(* USED TO LATCH A BIT TO CLEAR DATA AFTER UPSTACK TEST MODE IS OFF *)
IF 	csp_transfer_upstacker_sensors.debug_active
THEN
	debug_active_bool := TRUE;
END_IF

IF 	debug_active_bool
	AND NOT csp_transfer_upstacker_sensors.debug_active
THEN
	debug_active_clear := TRUE;
	debug_active_bool := FALSE;
END_IF

dry_cycle_ftrig(CLK :=csp_case_main_services.dry_cycle_mode); // falling edge of dry cycle mode, clear upstacker counts on completion of dry cycle mode. 
cleanout_mode_ftrig(CLK :=csp_main_motorization.empty_command); // falling edge of clean out mode, clear upstacker counts on completion of dry cycle mode. 


(* CLEARS SHIFT REGISTER BITS DURING SIZE CHANGE *)
IF 	csp_main_accuchange.machine_empty
	OR debug_active_clear
	OR process_message_is_on(csp_case_virtualMaster.runout_complete)
	OR dry_cycle_ftrig.Q
	OR cleanout_mode_ftrig.Q
THEN
	stack_count := 0;
	stack_made := FALSE;
	stack_on_way_to_loader := FALSE;
	stack_at_loader := FALSE;
	First_cycle_after_dry := TRUE;
	debug_active_clear := FALSE;
END_IF

//Resets First_Cycle_After_Dry

IF 	First_Cycle_After_Dry
	AND csp_main_motorization_virtualManager.axis.actual_position > 355
	AND csp_main_motorization_virtualManager.axis.actual_position < 359
THEN
	First_Cycle_After_Dry := False;
END_IF


(* CLEARS STACK AT LOADER AND ON WAY TO LOADER IF CROSSPUSHER REJECT *)
IF 	csp_transfer_crosspusher.reject_running
THEN
	stack_on_way_to_loader := FALSE;
	stack_at_loader := FALSE;
END_IF


(* MANUAL REMOVAL OF STACK AT UPSTACKER *)
IF 	stack_removed_from_upstack_cbtn.value_from_hmi = HMI_BUTTON_STATUS_ON//command_button_is_pressed(stack_removed_from_upstack_cbtn) 
THEN
	stack_removed_from_upstack := TRUE;
ELSE
	stack_removed_from_upstack := FALSE;
END_IF

IF stack_removed_from_upstack
THEN
	stack_count := 0;
END_IF


(* CHECKS STACK COUNT AGAINST CASE PATTERN COUNT TO KNOW IF STACK IS MADE *)
IF 	stack_count >= csp_main_brand.case_pattern.case_pattern_W
	OR stack_made_test
THEN 
	stack_made := TRUE;
ELSE
	stack_made := FALSE;
END_IF


(* CLEARS STACK MADE WHEN CORSSPUSHER RUNS TO LOAD - SAVES STACK AT LOADER VARIABLE FOR LOADER*)
IF 	stack_made
	AND csp_transfer_crosspusher_horizontal.active_cam = TRANSFER_CROSSPUSHER_HORIZONTAL_TO_LOAD
THEN
	stack_count := 0;
	stack_on_way_to_loader := TRUE;
END_IF


(* LOADER TRIGGER *)
IF 	test_loader_enable
	AND stack_on_way_to_loader (* STACK HAS BEEN PUSHED FROM UPSTACKER TO LOAD *)
	AND csp_transfer_crosspusher.loader_clear (* LOADER IS CLEAR *)
	AND csp_transfer_crosspusher_horizontal.at_load (* HORIZONTAL AT LOAD *)
	AND ABS(csp_transfer_crosspusher_follower.axis.actual_position - csp_transfer_crosspusher_follower.slave_scaling) < 2 (* FOLLOWER AT LOAD *)
	AND NOT csp_transfer_crosspusher_sensors.reject_stack (* NOT REJECT STACK *)
	AND NOT csp_transfer_crosspusher_sensors.no_load_bool.status (* NOT NO LOAD *)
	AND NOT csp_transfer_upstacker_sensors.debug_active
THEN
	//ITEM_HAS_TRANSFER_LOAD_BUILD_COMPLETE;
	;
END_IF


(* CLEARS STACK AT LOADER WHEN LOADER RUNS RUN CAM *)
clear_pos_stack_at_loader := csp_case_loader_pusher.slave_scaling - 15;

IF 	stack_on_way_to_loader
	AND csp_transfer_crosspusher_horizontal.at_load
	AND NOT csp_transfer_crosspusher_sensors.reject_stack (* NOT REJECT STACK *)
	AND NOT csp_transfer_crosspusher_sensors.no_load_bool.status (* NOT NO LOAD *)
THEN
	stack_at_loader := TRUE;
	stack_on_way_to_loader := FALSE;
END_IF

IF 	csp_case_loader_pusher.axis.actual_position > clear_pos_stack_at_loader
	AND stack_at_loader
THEN
	stack_in_case_at_loader := TRUE;
	stack_at_loader := FALSE;
END_IF


IF 	(csp_case_transport_ls_trailing.axis.actual_position > 60)
	AND (csp_case_transport_ls_trailing.axis.actual_position < 300)
THEN
	stack_in_case_at_loader := FALSE;
END_IF

(* MANUAL REMOVAL OF CASES AT LOADER*)
IF 	command_button_is_pressed(csp_case_loader.case_removed_at_loader_cbtn)
   	AND csp_transfer_upstacker.stack_in_case_at_loader
THEN
   csp_transfer_upstacker.stack_in_case_at_loader := FALSE;
END_IF


IF 	stack_in_case_at_loader
THEN
	boolean_set(stack_in_case_at_loader_boolean);
ELSE
	boolean_reset(stack_in_case_at_loader_boolean);
END_IF


(************************************************************************)

_handle_messages();

_write_output();

ACTION _handle_messages:
;
END_ACTION

ACTION _handle_process_test:
;
END_ACTION

ACTION _mode_manager:
IF process_mode_req_is_pending(prc)
THEN
    process_apply_mode_req_first_step(prc);
    CASE process_get_mode(prc) OF
        MODE_TO_ABSENT:
			;
        MODE_TO_INACTIVE:
			;
        MODE_TO_TEST:
			;
        MODE_TO_OPERATIONAL:
			;
    END_CASE
    process_apply_mode_req_second_step(prc);
END_IF
END_ACTION

ACTION _object_manager:
IF objects_initialization()
THEN
	sub_process_init(
		object_name					:= 'csp_transfer_upstacker.prc', 
		process						:= csp_transfer.prc, 
		CONVERSION_this				:= prc);
		
	prc_path 						:= process_get_path(prc);
	
	
	phase_generator_init(
		object_name					:= CONCAT(prc_path, '_phgen'), 
		modulo						:= 360, 
		resolution					:= PHASE_GENERATOR_RESOLUTION_UNIT, 
		axis						:= csp_transfer_upstacker_virtualMaster.axis, 
		process						:= prc, 
		CONVERSION_this				:= phgen);
		
	phase_init(
        object_name 				:= CONCAT(prc_path, '_cam_check_ph'),
        phase 						:= 0,	//Set at runtime!
        delay 						:= 0,
        max_compensation 			:= 0,
        generator 					:= phgen,
        process 					:= prc,
        CONVERSION_this 			:= cam_check_ph);
		
		
	command_button_init(
	    object_name 				:= CONCAT(prc_path, '_stack_removed_from_upstack_cbtn'),
	    process 					:= prc,
	    CONVERSION_this 			:= stack_removed_from_upstack_cbtn);
	
	
END_IF

IF objects_running()
THEN
	process_cycle(prc);
	
	phase_generator_cycle(phgen);
	phase_cycle(cam_check_ph);
END_IF
END_ACTION

ACTION _read_process_image:
;
END_ACTION

ACTION _read_var_input:
;
END_ACTION

ACTION _set_runtime_properties:
;
END_ACTION

ACTION _write_output:
;
END_ACTION

END_PROGRAM

// ---- Application/CSP/Transfer/Accumulator/Vitual Master/csp_transfer_accumulator_virtualMaster.TcPOU
(*********************************** G.D S.p.A. - Technical Department ***********************************
============= PROGRAM INFO ============
FOLDER:             TBD
MACHINES INVOLVED:  TBD 

============= DESCRIPTION =============
csp machine declaration

============= REVISIONS ===============
Date		Version	 	Author      	Description             
----------	-------		------------  	--------------------------------------------
2019/04/05 	0000.00	 	M.Grasso		Creation of the PRG

**********************************************************************************************************)
(*$R process_ref := prc; $*)
PROGRAM csp_transfer_accumulator_virtualMaster
VAR
	
	prc:											process;
	prc_path:										STRING;
	
	axis: 											axis;
	axis_actual_position:							LREAL;
	phgen:											phase_generator;
	
	disable_req:									BOOL;
	debug_state_machine:							BOOL := FALSE;
	debug_phase_machine_one_step:					BOOL := FALSE;
	debug_connection_machine_one_step:				BOOL := FALSE;
	
	phase_status: 									csp_transfer_accumulator_belt_phase_status_enum;
	phase_status_next: 								csp_transfer_accumulator_belt_phase_status_enum;
	phase_done: 									BOOL;
	phase_running: 									BOOL;
	phase_error:									BOOL;
	phase_time_out_tmr:								timer;
	phase_faulted_aem:	 							message;
	phase_conditions:								BOOL;
	
	connection_status: 								csp_transfer_accumulator_connection_status_enum;
	connection_status_next: 						csp_transfer_accumulator_connection_status_enum;
	connection_done: 								BOOL;
	connection_running: 							BOOL;
	connection_error:								BOOL;
	connection_time_out_tmr:						timer;
	connection_faulted_aem:	 						message;
	connection_conditions:							BOOL;
	connection_done_motcond:						motorization_conditioner;
	connection_motorization_moving:					BOOL;
	
	
	slave_scaling:									LREAL := 1.0 (*360.0*);
	master_scaling:									LREAL := 1.0 (*360.0*);

	home_position_master_offset_deg:				LREAL := 0.0;
	axis_calculate_cam_slave_master_position_deg:	LREAL := 0.0;
	axis_calculated_cam_slave_position_deg:			LREAL := 0.0;	
	slave_position_has_been_calculated:				BOOL  := FALSE;
	
	phase_velocity_degps:							LREAL := 100.0;
	engage_enable:									BOOL := TRUE;
	
END_VAR

VAR CONSTANT
			
	MOTOR_PHASE_POSITION_DEG:						LREAL := 60;
	MOTOR_PHASE_VELOCITY_DEGPS:						LREAL := 10;
	
	MOTOR_MAX_VELOCITY_DEGPS:						LREAL := 9600;
	MOTOR_MAX_ACCELERATION_DEGPS2:					LREAL := 48000;
	MOTOR_MAX_DECELERATION_DEGPS2:					LREAL := 48000;
	MOTOR_MAX_JERK_DEGPS3:							LREAL := 1000000; 
	MOTOR_MAX_FOLLOWING_ERROR_DEG:					LREAL := 2;
		
END_VAR

_read_var_input();

_object_manager();

IF 	NOT objects_running()
THEN
	RETURN;	
END_IF

_read_process_image();

_mode_manager();

CASE process_get_mode(prc) of
	MODE_ABSENT,
	MODE_INACTIVE:
		RETURN;
	MODE_TEST:
		_handle_process_test();
END_CASE

_set_runtime_properties();

(********************************* BODY *********************************)

IF connection_done
THEN 
	motorization_conditioner_start_done(connection_done_motcond);
END_IF

slave_scaling := csp_main_brand.case_pattern.case_pattern_W;

jog_manager_set_all_slave_axis_engaged(
	index					:= JOG_LIST_TRANSFER_ACCUMULATOR_VIRTUAL, 
	all_slave_axis_engaged	:= 	axis_is_cam_engaged(csp_transfer_upstacker_virtualMaster.axis)
							 	AND
							 	axis_is_cam_engaged(csp_transfer_accumulator_belt.axis),
	CONVERSION_this			:= csp_main_jogManager.jog_manager_virtual);

(* DISABLES VIRTUAL IS ANY OF THE SLAVES FAULT *)
IF NOT axis_is_disabled(axis)
	AND NOT axis_is_ok(FALSE, csp_transfer_accumulator_belt.axis)
	AND NOT axis_is_ok(FALSE, csp_transfer_upstacker_virtualMaster.axis)
THEN
	axis_disable(axis);
END_IF

(* RESETS AXES IF PHASE DONE AND CONNECTION DONE AND DISABLED *)
IF phase_done
	AND connection_done
	AND axis_is_disabled(axis)
THEN
	phase_done := FALSE;
	connection_done := FALSE;
END_IF

(* CLEARS PHASE AND CONNECTION ERRORS ON STOP *)
IF machine_is_stopped(csp.mch)
	OR machine_is_stop_emergency_active(csp.mch)
THEN
	phase_error := FALSE;
	connection_error := FALSE;
END_IF

phase();
connection();

(************************************************************************)

_handle_messages();

_write_output();

ACTION _handle_messages:
;
END_ACTION

ACTION _handle_process_test:
;
END_ACTION

ACTION _mode_manager:
IF process_mode_req_is_pending(prc)
THEN
    process_apply_mode_req_first_step(prc);
    CASE process_get_mode(prc) OF
        MODE_TO_ABSENT:
			;
        MODE_TO_INACTIVE:
			;
        MODE_TO_TEST:
			;
        MODE_TO_OPERATIONAL:
			;
    END_CASE
    process_apply_mode_req_second_step(prc);
END_IF
END_ACTION

ACTION _object_manager:
IF objects_initialization()
THEN	
	sub_process_init(
		object_name					:= 'csp_transfer_accumulator_virtualMaster.prc', 
		process						:= csp_transfer_accumulator.prc, 
		CONVERSION_this				:= prc);
		
	prc_path 						:= process_get_path(prc);
	
	axis_init(
		object_name					:= CONCAT(prc_path, '_axis'), 
		axis_type					:= AXIS_TYPE_VIRTUAL, 
		encoder_scaling_factor		:= G_VIRTUAL_ENCODER_SCALING_FACTOR_DEGPINC,
		modulo						:= G_MODULO_360_DEG, 
		process						:= prc, 
		CONVERSION_this				:= axis);
	
	axis_set_max_dynamic(
		reference_velocity			:=	MOTOR_MAX_VELOCITY_DEGPS,
		velocity					:=	MOTOR_MAX_VELOCITY_DEGPS,
		acceleration				:=	MOTOR_MAX_ACCELERATION_DEGPS2,
		deceleration				:=	MOTOR_MAX_DECELERATION_DEGPS2,
		jerk						:=	MOTOR_MAX_JERK_DEGPS3,
		following_error				:=	MOTOR_MAX_FOLLOWING_ERROR_DEG,
		CONVERSION_this				:=	axis);
		
	process_message_init(
		object_name					:=	CONCAT(prc_path, '_phase_faulted_aem'), 
		behaviour					:=	MESSAGE_BEHAVIOUR_EVENT,
		reset_timeout				:=	0,
		disableable					:=	TRUE,
		individual_reset			:=	FALSE,
		machine_reaction			:=	MACHINE_REACTION_NORMAL_STOP,
		typology					:=	MESSAGE_TYPOLOGY_ABNORMAL,
		process						:=	prc,
		CONVERSION_this				:=	phase_faulted_aem);
	
	timer_init(
		object_name					:= CONCAT(prc_path, 'phase_time_out_tmr'),
		process						:= prc,
		CONVERSION_this				:= phase_time_out_tmr);
	
	process_message_init(
		object_name					:=	CONCAT(prc_path, '_connection_faulted_aem'), 
		behaviour					:=	MESSAGE_BEHAVIOUR_EVENT,
		reset_timeout				:=	0,
		disableable					:=	TRUE,
		individual_reset			:=	FALSE,
		machine_reaction			:=	MACHINE_REACTION_NORMAL_STOP,
		typology					:=	MESSAGE_TYPOLOGY_ABNORMAL,
		process						:=	prc,
		CONVERSION_this				:=	connection_faulted_aem);
	
	timer_init(
		object_name					:= CONCAT(prc_path, 'connection_time_out_tmr'),
		process						:= prc,
		CONVERSION_this				:= connection_time_out_tmr);
				 
	phase_generator_init(
		object_name					:= CONCAT(prc_path, '_phgen'), 
		modulo						:= 360, 
		resolution					:= PHASE_GENERATOR_RESOLUTION_UNIT, 
		axis						:= axis, 
		process						:= prc, 
		CONVERSION_this				:= phgen);
		
	motorization_conditioner_init(
		object_name					:=	CONCAT(prc_path, 'connection_done_motcond'),
		velocity_limit				:=	0.0,
		velocity_limit_active		:=	FALSE,
		idle_handshake_active		:=	FALSE,
		execute_handshake_active	:=	TRUE,
		hold_handshake_active		:=	FALSE,
		suspend_handshake_active	:=	FALSE,
		complete_handshake_active	:=	FALSE,
		abort_handshake_active		:=	FALSE,
		stop_handshake_active		:=	FALSE,
		origin						:=	MOTORIZATION_CONDITIONER_ORIGIN_INTERNAL,
		manager						:=	csp_main_motorization_manager.motm,
		process						:=	prc,
		CONVERSION_this				:=	connection_done_motcond);

		
	jog_manager_add_axis(
		list_index					:= JOG_LIST_TRANSFER_ACCUMULATOR_VIRTUAL,
		axis						:= axis,
		master_axis					:= TRUE,
		jog_type					:= JOG_TYPE_ROTATIVE_PLUS,
		sw_limit_positive			:= 0,
		sw_limit_negative			:= 0,
		CONVERSION_this				:= csp_main_jogManager.jog_manager_virtual);
END_IF

IF objects_running()
THEN
	process_cycle(prc);
	motorization_conditioner_cycle(connection_done_motcond);
	
	axis_cycle(axis);
	phase_generator_cycle(phgen);		
END_IF
END_ACTION

ACTION _read_process_image:
;
END_ACTION

ACTION _read_var_input:
disable_req := csp_transfer.virtual_disable_req;
END_ACTION

ACTION _set_runtime_properties:
axis_actual_position := axis_get_actual_modulo_position(axis);
END_ACTION

ACTION _write_output:
;
END_ACTION

ACTION connection:
connection_conditions :=	
	axis_is_ok(FALSE, axis)
	AND 
	NOT process_message_is_on(connection_faulted_aem)
	AND
	phase_done;

(* connection_done reset *)
IF	connection_done
	AND	
	NOT connection_conditions
THEN
	connection_done := FALSE;
END_IF

(* Exit conditions *)
IF	NOT connection_conditions
	AND
	NOT motorization_manager_is_stopping(csp_main_motorization_manager.motm)	
THEN	
	connection_status_next := CSP_TRANSFER_ACCUMULATOR_STATUS_CONNECTION_ERROR;
	connection_status := connection_status_next;	
END_IF

(*************** MACHINE STATUS ***************)
CASE connection_status OF

	CSP_TRANSFER_ACCUMULATOR_STATUS_CONNECTION_START:	(* Start connection *)
	
		IF	motorization_manager_is_starting(csp_main_motorization_manager.motm) //TODOPZ: da decidere a che livello usare le variabili di i e o: wn_feeding.i_motorization_is_starting?					
		THEN
			connection_running := TRUE;
			connection_status_next := CSP_TRANSFER_ACCUMULATOR_STATUS_CONNECTION_ENGAGE;
		END_IF
		
	CSP_TRANSFER_ACCUMULATOR_STATUS_CONNECTION_ENGAGE:	

		axis_engage_cam(
			cam_id							:=	FORWARD_CAM,	
			master_engage_mode				:=	AXIS_CAM_ENGAGE_RELATIVE,
			slave_engage_mode				:=	AXIS_CAM_ENGAGE_RELATIVE,
			activation_mode					:=	AXIS_CAM_ACTIVATION_IMMEDIATELY,
			activation_position				:=	0.0,
			master_scaling_mode				:=	AXIS_CAM_SCALING_MODE_USER_DEFINED,
			slave_scaling_mode				:=	AXIS_CAM_SCALING_MODE_AUTOOFFSET,
			master_offset					:=	0.0, 
			slave_offset					:=	0.0,
			master_scaling					:=	master_scaling,
			slave_scaling					:=	slave_scaling,
			interpolation_type				:=	AXIS_CAM_INTERPOLATION_SPLINE,	 
			master							:=	csp_transfer_virtualMaster.axis,
			CONVERSION_this					:=	axis);
		
		connection_status_next:= CSP_TRANSFER_ACCUMULATOR_STATUS_CONNECTION_ENGAGED;
	
		
	CSP_TRANSFER_ACCUMULATOR_STATUS_CONNECTION_ENGAGED:
	
		IF 	axis_is_cam_engaged(axis) 
		THEN				
			connection_status_next:= CSP_TRANSFER_ACCUMULATOR_STATUS_CONNECTION_DONE;			
		END_IF
	
			
	CSP_TRANSFER_ACCUMULATOR_STATUS_CONNECTION_DONE:	(* Connection done *)	
	
		connection_running := FALSE;
		connection_done := TRUE;
		IF	motorization_manager_is_starting(csp_main_motorization_manager.motm)
		THEN
			motorization_conditioner_start_done(connection_done_motcond);
		END_IF
			
	
	CSP_TRANSFER_ACCUMULATOR_STATUS_CONNECTION_ERROR:	(* Connection error *)	
	
		IF 	connection_running
			OR NOT axis_is_ok(FALSE, axis)
		THEN
			axis_disable(axis);
			connection_error := TRUE;							
		END_IF
		connection_running	:= FALSE;
		connection_done 	:= FALSE;	
		
		IF	connection_conditions
		THEN		
			connection_status_next := CSP_TRANSFER_ACCUMULATOR_STATUS_CONNECTION_START;
		END_IF
		
END_CASE

IF 	NOT debug_state_machine
	OR
	debug_connection_machine_one_step	
THEN
	connection_status := connection_status_next;
	debug_connection_machine_one_step := FALSE;
END_IF

connection_motorization_moving	:= 
	motorization_manager_is_starting(csp_main_motorization_manager.motm)
	OR
	motorization_manager_is_execute(csp_main_motorization_manager.motm)
	OR
	motorization_manager_is_stopping(csp_main_motorization_manager.motm)
	OR
	motorization_manager_is_suspended(csp_main_motorization_manager.motm)
	OR
	motorization_manager_is_suspending(csp_main_motorization_manager.motm)
	OR
	motorization_manager_is_unsuspending(csp_main_motorization_manager.motm)
	OR 
	motorization_manager_is_holding(csp_main_motorization_manager.motm)
	OR
	motorization_manager_is_held(csp_main_motorization_manager.motm)
	OR
	motorization_manager_is_unholding(csp_main_motorization_manager.motm);	
	
(* Connection timeout *)
IF	(connection_running
AND NOT debug_state_machine)	
OR connection_error
THEN
	IF	timer_is_expired(connection_time_out_tmr)
	THEN
		process_message_set(1, connection_status, 0, connection_faulted_aem);
	END_IF
ELSE
	timer_restart(10000, connection_time_out_tmr);
END_IF
END_ACTION

ACTION phase:
phase_conditions :=
	axis_is_ok(FALSE, axis)
	AND
	process_is_ready(prc)
	AND
	process_subtree_is_ready(prc)
	AND
	NOT jog_manager_is_jog_axis_active(JOG_LIST_TRANSFER_ACCUMULATOR_VIRTUAL, csp_main_jogManager.jog_manager_virtual)
	AND				
	NOT csp_transfer_main_brand.cam_data_changed
	AND
	NOT disable_req;		
	
(* phase_done reset *)
IF	phase_done
	AND
	NOT phase_conditions
THEN
	phase_done:= FALSE;
END_IF

(* Exit condition *)
IF 	NOT phase_conditions
THEN
	phase_status_next := CSP_TRANSFER_ACCUMULATOR_BELT_STATUS_PHASE_ERROR;
	phase_status := phase_status_next;	
END_IF

(*************** MACHINE STATUS ***************)
CASE phase_status OF

	CSP_TRANSFER_ACCUMULATOR_BELT_STATUS_PHASE_START:	(* Start phasing *)
		IF	motorization_manager_is_starting(csp_main_motorization_manager.motm) 					
			AND csp_transfer_virtualMaster.phase_done
			AND csp_transfer_virtualMaster.connection_done
		THEN
			phase_running := TRUE;			
			phase_status_next := CSP_TRANSFER_ACCUMULATOR_BELT_STATUS_PHASE_DISABLE;
		END_IF
						
	CSP_TRANSFER_ACCUMULATOR_BELT_STATUS_PHASE_DISABLE:
	
		axis_disable(axis);		
		
		IF 	axis_is_disabled(axis)
		THEN
			phase_status_next := CSP_TRANSFER_ACCUMULATOR_BELT_STATUS_PHASE_ENABLE;
		END_IF
		
		
	CSP_TRANSFER_ACCUMULATOR_BELT_STATUS_PHASE_ENABLE:
	
		axis_enable(axis);
		
		IF 	axis_is_enabled(axis)
		THEN
			phase_status_next := CSP_TRANSFER_ACCUMULATOR_BELT_STATUS_PHASE_ENABLED;
		END_IF
		
		
	CSP_TRANSFER_ACCUMULATOR_BELT_STATUS_PHASE_ENABLED:
	
		IF 	axis_is_standstill(axis) 
		THEN
			phase_status_next := CSP_TRANSFER_ACCUMULATOR_BELT_STATUS_PHASE_CALCULATE_SLAVE_POSITION_REQUEST;								
		END_IF
		
		
	CSP_TRANSFER_ACCUMULATOR_BELT_STATUS_PHASE_CALCULATE_SLAVE_POSITION_REQUEST:
	
		slave_position_has_been_calculated := FALSE;
	
		(* Gets the position of the master axis *)
		axis_calculate_cam_slave_master_position_deg := 
			LMOD(axis_get_actual_modulo_position(csp_transfer_virtualMaster.axis)
			+ home_position_master_offset_deg, G_MODULO_360_DEG);
			
		(* Gets cam data for slave axis to master *)
		IF axis_calculate_cam_slave_dynamics_data(
			cam_id := FORWARD_CAM,
			master_scaling := master_scaling,
			master_position := axis_calculate_cam_slave_master_position_deg,
			slave_scaling := slave_scaling,
			CONVERSION_this := axis)
			THEN
				phase_status_next := CSP_TRANSFER_ACCUMULATOR_BELT_STATUS_PHASE_CALCULATING_SLAVE_POSITION;
		END_IF
	
		
	CSP_TRANSFER_ACCUMULATOR_BELT_STATUS_PHASE_CALCULATING_SLAVE_POSITION:
	
		IF axis_cam_slave_dynamics_data_calculated(axis)
		THEN
			axis_calculated_cam_slave_position_deg := axis_get_cam_slave_dynamics_position(axis);
			slave_position_has_been_calculated := TRUE;
			phase_status_next := CSP_TRANSFER_ACCUMULATOR_BELT_STATUS_PHASE_REQUESTED;
		END_IF
	
	
	CSP_TRANSFER_ACCUMULATOR_BELT_STATUS_PHASE_REQUESTED:
	
		IF	axis_is_standstill(axis)
		THEN
		 axis_move_absolute(
			position 		:= axis_calculated_cam_slave_position_deg,
			velocity 		:= phase_velocity_degps,
			direction		:= AXIS_SHORTEST_WAY,
			acceleration 	:= MOTOR_MAX_ACCELERATION_DEGPS2,
			deceleration 	:= MOTOR_MAX_DECELERATION_DEGPS2, 
			jerk 			:= MOTOR_MAX_JERK_DEGPS3, 
			buffer_mode 	:= AXIS_BUFFER_MODE_BUFFERED,
			CONVERSION_this := axis
			); 			
		END_IF

		IF axis_is_absolute_moving(axis)
		THEN
			phase_status_next	:=	CSP_TRANSFER_ACCUMULATOR_BELT_STATUS_PHASE_PHASING;
		END_IF
	
		
	CSP_TRANSFER_ACCUMULATOR_BELT_STATUS_PHASE_PHASING:
	
		IF axis_is_standstill(axis)
		THEN
			phase_status_next	:=	CSP_TRANSFER_ACCUMULATOR_BELT_STATUS_PHASE_PHASED;
		END_IF
		
		
	CSP_TRANSFER_ACCUMULATOR_BELT_STATUS_PHASE_PHASED:
	
		IF engage_enable
		THEN
			phase_status_next := CSP_TRANSFER_ACCUMULATOR_BELT_STATUS_PHASE_DONE;
		END_IF
		
		
	CSP_TRANSFER_ACCUMULATOR_BELT_STATUS_PHASE_DONE:	(* Phase done *)
			
		phase_running := FALSE;
		phase_done := TRUE;		

		IF NOT axis_is_enabled(axis)
		THEN
				phase_status_next := CSP_TRANSFER_ACCUMULATOR_BELT_STATUS_PHASE_ERROR;
		END_IF		
	
		
	CSP_TRANSFER_ACCUMULATOR_BELT_STATUS_PHASE_ERROR:	(* Phase error *)
	
		IF	phase_running
			OR NOT axis_is_ok(FALSE, axis)
		THEN
			phase_error := TRUE;
			axis_disable(axis);									
		END_IF
		phase_running := FALSE;
		
		IF	phase_conditions 	
		THEN
			phase_status_next := CSP_TRANSFER_ACCUMULATOR_BELT_STATUS_PHASE_START;
		END_IF
		
END_CASE

IF 	NOT debug_state_machine
	OR
	debug_phase_machine_one_step	
THEN
	phase_status := phase_status_next;
	debug_phase_machine_one_step := FALSE;
END_IF

(* Phasing timeout *)
IF (phase_running
	AND NOT debug_state_machine)
	OR phase_error
THEN
	IF	timer_is_expired(phase_time_out_tmr)
	THEN
		process_message_set(1, phase_status, 0, phase_faulted_aem);
	END_IF
ELSE
	timer_restart(30000, phase_time_out_tmr);
END_IF
END_ACTION

END_PROGRAM

// ---- Application/CSP/Main/Brand/csp_main_brand.TcPOU
(*********************************** G.D S.p.A. - Technical Department ***********************************
============= PROGRAM INFO ============
FOLDER:             TBD
MACHINES INVOLVED:  TBD 

============= DESCRIPTION =============
csp brand management program

============= REVISIONS ===============
Date		Version	 	Author      	Description             
----------	-------		------------  	--------------------------------------------
2019/04/05 	0000.00	 	M.Grasso		Creation of the PRG

**********************************************************************************************************)
(*$R
	process_ref := prc;
$*)
PROGRAM csp_main_brand
VAR
	prc:														process;
	prc_path:													STRING;

	p_carton_format:											csp_main_brand_carton_format_enum;	(*$P $*)
	
	carton_dimension:											csp_main_brand_product_dimension;
	
	case_pattern:												csp_main_brand_case_pattern;

	nominal_case_rate_ppm:										LREAL := 15.63; (*$P $*)
	surge_case_rate_ppm:										LREAL := 17.19; (*$P $*)
	
	cartons_per_minute:											INT := 63;
	
	cups_number_for_carton:										INT	:=	24;	
	infeed_reject_use_both_sides:								BOOL := FALSE; (*$P $*)
	Rollover_Carton:											BOOL := TRUE; (*$P $*)
	carton_belts_tooth_distance_mm:								LREAL := 150;
	choice:														DINT :=1;
	
	metering_carton_gap:										LREAL; (*$P $*)
	post_waterfall_carton_gap:									LREAL; (*$P $*)
	
	count_changed:												BOOL;
	
	count:														STRING := 'First Start'; (*$P $*)
	count_old:													STRING := 'First Start'; (*$P $*)
	count_old_po:												parameter_overwrite;
	
	cam_data_changed:											BOOL;			
	Cartons_per_case: 											INT;
END_VAR

_read_var_input();

_object_manager();

IF NOT objects_running()
THEN
	RETURN;	
END_IF

_read_process_image();

_mode_manager();

CASE process_get_mode(prc) OF
	MODE_ABSENT,
	MODE_INACTIVE:
		RETURN;
	MODE_TEST:
		_handle_process_test();
END_CASE

_set_runtime_properties();

(********************************* BODY *********************************)



(************************************************************************)

IF	(
		count_old
		<>
		count
	)
	AND
	(
		count <> ''
	)
THEN		
	count_old := count;
	count_changed := TRUE;
END_IF

IF csp_main_accuChange.Brand_Change_Occurred 
THEN 
	count_changed := FALSE;
END_IF


IF 	p_carton_format = csp_MAIN_BRAND_16_COUNT_2x3CARTON_4_COUNT_CASE
	OR
	p_carton_format = csp_MAIN_BRAND_18_COUNT_2x3CARTON_4_COUNT_CASE
	OR
	p_carton_format = csp_MAIN_BRAND_20_COUNT_2x4CARTON_4_COUNT_CASE	
	OR
	p_carton_format = csp_MAIN_BRAND_22_COUNT_2x4CARTON_4_COUNT_CASE
	OR
	p_carton_format = csp_MAIN_BRAND_24_COUNT_2x4CARTON_4_COUNT_CASE	
	OR
	p_carton_format = csp_MAIN_BRAND_28_COUNT_2x4CARTON_4_COUNT_CASE	
	OR
	p_carton_format = csp_MAIN_BRAND_30_COUNT_2x4CARTON_4_COUNT_CASE
	OR	
	p_carton_format = csp_MAIN_BRAND_32_COUNT_2x4CARTON_4_COUNT_CASE
	OR
	p_carton_format = csp_MAIN_BRAND_34_COUNT_3x4CARTON_4_COUNT_CASE
	OR	
	p_carton_format = csp_MAIN_BRAND_36_COUNT_3x4CARTON_4_COUNT_CASE
	OR	
	p_carton_format = csp_MAIN_BRAND_44_COUNT_3x4CARTON_4_COUNT_CASE
	OR
	p_carton_format = csp_MAIN_BRAND_46_COUNT_3x4CARTON_4_COUNT_CASE
	OR
	p_carton_format = csp_MAIN_BRAND_48_COUNT_3x4CARTON_4_COUNT_CASE
	OR
	count = '32Count'
	OR
	count = '24Count'
	THEN
		Cartons_per_case := 4;
	ELSE
		Cartons_per_case := 6;
END_IF
(************************************************************************)

_handle_messages();

_write_output();

ACTION _handle_messages:
;
END_ACTION

ACTION _handle_process_test:
;
END_ACTION

ACTION _mode_manager:
IF process_mode_req_is_pending(prc)
THEN
    process_apply_mode_req_first_step(prc);
    CASE process_get_mode(prc) OF
        MODE_TO_ABSENT:
			;
        MODE_TO_INACTIVE:
			;
        MODE_TO_TEST:
			;
        MODE_TO_OPERATIONAL:
			;
    END_CASE
    process_apply_mode_req_second_step(prc);
END_IF
END_ACTION

ACTION _object_manager:
IF objects_initialization()
THEN
	sub_process_init(
		object_name					:= 'csp_main_brand.prc', 
		process						:= csp_main.prc, 
		CONVERSION_this				:= prc);
		
	prc_path 						:= process_get_path(prc);


	
parameter_overwrite_string_init(
        object_name:= 'csp_main_brand.count_old_po',
        size_of_parameter:= SIZEOF(count_old),
        parameter:= count_old,
        process:= prc,
        CONVERSION_this:= count_old_po);	
END_IF

IF objects_running()
THEN
	process_cycle(prc);
END_IF
END_ACTION

ACTION _read_process_image:
;
END_ACTION

ACTION _read_var_input:
;
END_ACTION

ACTION _set_runtime_properties:
;
END_ACTION

ACTION _write_output:
;
END_ACTION

END_PROGRAM

// ---- POUs/AFL extensions/jog_manager/commands/jog_manager_set_all_slave_axis_engaged.TcPOU
(*$
	Set the all slave axis engaged condition <b><i>this</i></b>.
	The method returns <i>TRUE</i> if the command is accepted, otherwise it returns <i>FALSE</i>.
$*)
FUNCTION jog_manager_set_all_slave_axis_engaged : BOOL
VAR_INPUT
	index:					UINT;
	all_slave_axis_engaged:	BOOL;
END_VAR
VAR_IN_OUT
    CONVERSION_this:		jog_manager;	(*$ Instance to which the method applies $*)
END_VAR

IF	NOT (descriptor_mode_is_operational(CONVERSION_this.descriptor)
		(*OR
		descriptor_mode_is_test(CONVERSION_this.descriptor)*)
		OR
		(index <= JOG_MANAGER_JOG_LIST_NONE)
		OR
		(index > JOG_MANAGER_JOG_LIST_MAX))
THEN
	jog_manager_set_all_slave_axis_engaged := FALSE;				(* command rejected *)
 	RETURN;
END_IF

IF	(CONVERSION_this.axis_list[index].axis = G_framework.NULL)
	OR
	NOT CONVERSION_this.axis_list[index].master_axis 
THEN
	jog_manager_set_all_slave_axis_engaged := FALSE;				(* command rejected *)
 	RETURN;
END_IF

CONVERSION_this.axis_list[index].all_slave_axis_engaged := all_slave_axis_engaged;
jog_manager_set_all_slave_axis_engaged := TRUE;						(* command accepted *)

END_FUNCTION

// ---- Application/CSP/Transfer/Accumulator/Belt/csp_transfer_accumulator_belt.TcPOU
(*********************************** G.D S.p.A. - Technical Department ***********************************
============= PROGRAM INFO ============
FOLDER:             TBD
MACHINES INVOLVED:  TBD 

============= DESCRIPTION =============
csp machine declaration

============= REVISIONS ===============
Date		Version	 	Author      	Description             
----------	-------		------------  	--------------------------------------------
2019/04/05 	0000.00	 	M.Grasso		Creation of the PRG

**********************************************************************************************************)
(*$R process_ref := prc; $*)
PROGRAM csp_transfer_accumulator_belt
VAR
	
	prc:												process;
	prc_path:											STRING;
	
	axis:												axis;
	phase_position_deg:									LREAL := 0;
	phase_velocity_degps:								LREAL := 100.0;
		
	home_position_master_offset_deg:					LREAL := 0.0;
	axis_calculate_cam_slave_master_position_deg:		LREAL := 0.0;
	axis_calculated_cam_slave_position_deg:				LREAL := 0.0;	
	slave_position_has_been_calculated:					BOOL  := FALSE;
	
	phase_enable:										BOOL := TRUE;
	slave_position_request:								BOOL := TRUE;
	engage_enable:										BOOL := TRUE;
	debug_state_machine_one_step:						BOOL := FALSE;
	
	cam_id:												DINT  := FORWARD_CAM;
	master_position:									LREAL := 30;
	master_cam:											LREAL := 30;
	
	slave_offset:										LREAL := 0;
	
	axis_actual_position:								LREAL;
	
	disable_req:										BOOL;
	debug_state_machine:								BOOL := FALSE;
	debug_phase_machine_one_step:						BOOL := FALSE;
	debug_connection_machine_one_step:					BOOL := FALSE;
	
	phase_status: 										csp_transfer_accumulator_belt_phase_status_enum;
	phase_status_next: 									csp_transfer_accumulator_belt_phase_status_enum;
	phase_done: 										BOOL;
	phase_running: 										BOOL;
	phase_error:										BOOL;
	phase_time_out_tmr:									timer;
	phase_faulted_aem:	 								message;
	phase_conditions:									BOOL;
	phase_master_is_engaged:							BOOL;
	
	cam_change_check_ph:								phase;
	
	connection_status: 									csp_transfer_accumulator_connection_status_enum;
	connection_status_next: 							csp_transfer_accumulator_connection_status_enum;
	connection_done: 									BOOL;
	connection_running: 								BOOL;
	connection_error:									BOOL;
	connection_time_out_tmr:							timer;
	connection_faulted_aem:	 							message;
	connection_conditions:								BOOL;
	connection_done_motcond:							motorization_conditioner;
	connection_motorization_moving:						BOOL;
	
	run:												BOOL;
	dwell:												BOOL;
	
	run_test:											BOOL;
	dwell_test:											BOOL := TRUE;
		
	active_cam:											DINT := DWELL_CAM;
	next_cam:											DINT := DWELL_CAM;	
	master_offset:										LREAL := 0;
	master_scaling:										LREAL := 1.0;
	slave_scaling:										LREAL := 200;

	torque_limit:										INT := 500; (*$P $*)
	torque_limit_old:									INT;
	overrun_percentage:									LREAL := 10; (*$P $*)
	
	activation_mode:									axis_cam_activation_mode_enum;
	
	CAM_CHANGE_CHECK_DEG:								LREAL := 80; (*$P $*)
	
	servo_on_condition: 								BOOL;
	
	Startup_run_bost: 									LREAL := 1;
	Startup_run_bost_ton:                               TON;
	startup_bost_condition: 							BOOL;
	enable_delay: 										TON;
	Torque_force_constant: 								LREAL := 1.33;
	motor_backup: 										LREAL :=-6;	(*$P $*)
	motor_backed_up: 									BOOL := FALSE;
END_VAR

VAR CONSTANT
	(*Just in case you prefer having constants instead of numbers*)	
	G_MODULO_MM:										LREAL := 360;
	
	MOTOR_MAX_VELOCITY_DEGPS:							LREAL := 9600;
	MOTOR_MAX_ACCELLERATION_DEGPS2:						LREAL := 4800;
	MOTOR_MAX_DECELLERATION_DEGPS2:						LREAL := 4800;
	MOTOR_MAX_JERK_DEGPS3:								LREAL := 100000000; 
	MOTOR_MAX_FOLLOWING_ERROR_DEG:						LREAL := 2;
	
END_VAR

_read_var_input();

_object_manager();

IF 	NOT objects_running()
THEN
	RETURN;	
END_IF

_read_process_image();

_mode_manager();

CASE process_get_mode(prc) OF
	MODE_ABSENT:
		IF axis_get_mode(axis) = MODE_TEST
		THEN
			safety_integrated_series_close(csp_transfer_main_safety_drives_SD41300.chB_smes_sis);
		END_IF
		RETURN;
	MODE_INACTIVE:
		RETURN;
	MODE_TEST:
		_handle_process_test();
END_CASE

(********************************* BODY *********************************)
axis.actual_torque := (axis.actual_current * Torque_force_constant)/1000;

(* SET TORQUE LIMIT *)
IF torque_limit <> torque_limit_old
THEN
	IF soe_drive_channel_write_parameter(
		channel:= csp_transfer_accumulator_belt.axis.soe_drive_channel, 
		idn:= S_0_IDN + 92, 
		data_element:= soe_drive_element_value, 
		data_source:= ADR(torque_limit), 
		data_lenght:= SIZEOF(torque_limit),
		CONVERSION_this:= csp_transfer_accumulator_belt.axis.soe_drive^) = SOE_DRIVE_RETURN_VALUE_DONE
	THEN
		torque_limit_old := torque_limit;
	END_IF
END_IF

(* Connection Done Test - RMH *)
IF connection_done
THEN 
	motorization_conditioner_start_done(connection_done_motcond);
END_IF

(* SET CAM CHANGE FOR WHEN TO INDEX *)
phase_set_data(
	phase				:= CAM_CHANGE_CHECK_DEG,
	delay				:= 0,			
	max_compensation	:= 0,			
	CONVERSION_this		:= cam_change_check_ph);
	
IF phase_edge(cam_change_check_ph)
THEN		
	(* TO RUN *)
	IF run_test
		OR 
		(* LEVEL IS APPROPRIATE *)
		(
			csp_transfer_infeed_accumulation_level.level_status > CSP_TRANSFER_INFEED_ACCUMULATION_LEVEL_STATUS_UNDER_MIN
			OR
			csp_main_motorization.empty_command
		)
		(* CLAMPS ARE OPEN *)
		AND csp_transfer_infeed_clamp.clamp_open_bool
		(* CARTONS NOT AT BACKSTOP *)
		AND NOT csp_transfer_upstacker_sensors.carton_backstop_bool // BLOCKED BY FINGERS AT 80
		(* NOT IN REJECT *)
		AND NOT csp_transfer_crosspusher_sensors.reject_stack
		AND NOT csp_transfer_upstacker_sensors.dwell_transfer_empty
	THEN
		run := TRUE;
	ELSE
		dwell := TRUE;
	END_IF	
END_IF

(* Created startup timer to give the accumulator belt an additional scaling during start up to help drive product into the upstacker*)
Startup_run_bost_ton(IN:=csp.o_machine_is_running , PT:=T#3S , Q=> startup_bost_condition , ET=> );

IF NOT startup_bost_condition
THEN
	startup_run_bost := 1.5;
ELSE
	startup_run_bost := 1.0;	
END_IF

(* SET INDEX DISTANCE DYNAMICALLY BY SIZE OF CARTONS + DIMENSIONS + OVERRUN PERCENTAGE *)
slave_scaling := 	SEL(csp_main_brand.Rollover_Carton,
						csp_main_brand.carton_dimension.carton_size_W_mm, 
						csp_main_brand.carton_dimension.carton_size_L_mm) 
					* 
					csp_main_brand.case_pattern.case_pattern_L
					* 
					(1 + (overrun_percentage / 100))
					*
					Startup_run_bost; //At startup this is a multiplier to run the accumulator belt further to help get cases into the accumulator


(* ERROR HANDLING LOGIC TO CATCH CAM ERROR *)
IF active_cam = 0
THEN 
	active_cam := DWELL_CAM;
END_IF

(* RESETS AXES IF PHASE DONE AND CONNECTION DONE AND DISABLED *)
IF 	phase_done
	AND connection_done
	AND axis_is_disabled(axis)
THEN
	phase_done := FALSE;
	connection_done := FALSE;
END_IF

(* CLEARS CONNECTION AND PHASE ERRORS *)
IF	machine_is_stopped(csp.mch)
	OR machine_is_stop_emergency_active(csp.mch)
	OR machine_is_ready(csp.mch)
	OR csp_main_services_pushbuttons.i_reset_button
THEN
	phase_error := FALSE;
	connection_error := FALSE;	
END_IF

//Temp test on move back
IF	axis.actual_velocity <1 //axis_is_standstill(axis)
	AND NOT motor_backed_up
	AND	(next_cam = DWELL_CAM)
	AND NOT csp_main_motorization.empty_command
THEN
	axis_move_relative(
		distance:= motor_backup,
		velocity 		:= phase_velocity_degps,
		acceleration 	:= MOTOR_MAX_ACCELLERATION_DEGPS2,
		deceleration 	:= MOTOR_MAX_DECELLERATION_DEGPS2,
		jerk 			:= MOTOR_MAX_JERK_DEGPS3, 
		buffer_mode 	:= AXIS_BUFFER_MODE_ABORTING,
		CONVERSION_this := axis);
		
	motor_backed_up := TRUE;
END_IF

IF 	axis.actual_velocity >1//NOT axis_is_standstill(axis)
	AND motor_backed_up
	AND (active_cam = TRANSFER_ACCUMULATOR_BELT_RUN)
THEN
	motor_backed_up := FALSE;
END_IF

(* MAIN POU ACTIONS *)
phase();
connection();
_set_runtime_properties();

(************************************************************************)

_handle_messages();

_write_output();

ACTION _handle_messages:
;
END_ACTION

ACTION _handle_process_test:
;
END_ACTION

ACTION _mode_manager:
IF process_mode_req_is_pending(prc)
THEN
    process_apply_mode_req_first_step(prc);
    CASE process_get_mode(prc) OF
        MODE_TO_ABSENT:
			;
        MODE_TO_INACTIVE:
			;
        MODE_TO_TEST:
			;
        MODE_TO_OPERATIONAL:
			;
    END_CASE
    process_apply_mode_req_second_step(prc);
END_IF
END_ACTION

ACTION _object_manager:
IF objects_initialization()
THEN
	sub_process_init(
		object_name					:= 'csp_transfer_accumulator_belt.prc', 
		process						:= csp_transfer_accumulator.prc, 
		CONVERSION_this				:= prc);
		
	prc_path 						:= process_get_path(prc);
	
	axis_init(
		object_name					:= CONCAT(prc_path, '_axis'), 
		axis_type					:= AXIS_TYPE_SERVO, 
		encoder_scaling_factor		:= G_SERVO_ENCODER_SCALING_FACTOR_DEGPINC,
		modulo						:= G_MODULO_MM, 
		process						:= prc, 
		CONVERSION_this				:= axis);
		
	axis_init_absolute_encoder_preset(	
		position					:=	0,
		CONVERSION_this				:=	axis);	
	
	axis_set_max_dynamic(
		reference_velocity			:=	MOTOR_MAX_VELOCITY_DEGPS,
		velocity					:=	MOTOR_MAX_VELOCITY_DEGPS,
		acceleration				:=	MOTOR_MAX_ACCELLERATION_DEGPS2,
		deceleration				:=	MOTOR_MAX_DECELLERATION_DEGPS2,
		jerk						:=	MOTOR_MAX_JERK_DEGPS3,
		following_error				:=	MOTOR_MAX_FOLLOWING_ERROR_DEG,
		CONVERSION_this				:=	axis);

	jog_manager_add_axis(
		list_index					:= SMTR41323_TRANSFER_ACCUMULATOR_BELT,
		axis						:= axis,
		master_axis					:= FALSE,
		jog_type					:= JOG_TYPE_LINEAR_PLUS,
		sw_limit_positive			:= 0.0,
		sw_limit_negative			:= 0.0,
		CONVERSION_this				:= csp_main_jogManager.jog_manager_real);
		
	IF 	csp_main_configurator.Physical_hw
	THEN
		axis_add_safety_integrated_series(
			safety_integrated_series := csp_transfer_main_safety_drives_SD41300.chB_smes_sis,
			CONVERSION_this			:= axis);
	END_IF
		
	axis_add_soe_drive(
		channel						:=	SOE_DRIVE_CHANNEL_B,
		soe_drive					:=	csp_transfer_main_drives.SD41300_drv,
		CONVERSION_this				:=	axis);
		
	process_message_init(
		object_name					:=	CONCAT(prc_path, '_phase_faulted_aem'), 
		behaviour					:=	MESSAGE_BEHAVIOUR_EVENT,
		reset_timeout				:=	0,
		disableable					:=	TRUE,
		individual_reset			:=	FALSE,
		machine_reaction			:=	MACHINE_REACTION_NORMAL_STOP,
		typology					:=	MESSAGE_TYPOLOGY_ABNORMAL,
		process						:=	prc,
		CONVERSION_this				:=	phase_faulted_aem);
	
	timer_init(
		object_name					:= CONCAT(prc_path, 'phase_time_out_tmr'),
		process						:= prc,
		CONVERSION_this				:= phase_time_out_tmr);
	
	process_message_init(
		object_name					:=	CONCAT(prc_path, '_connection_faulted_aem'), 
		behaviour					:=	MESSAGE_BEHAVIOUR_EVENT,
		reset_timeout				:=	0,
		disableable					:=	TRUE,
		individual_reset			:=	FALSE,
		machine_reaction			:=	MACHINE_REACTION_NORMAL_STOP,
		typology					:=	MESSAGE_TYPOLOGY_ABNORMAL,
		process						:=	prc,
		CONVERSION_this				:=	connection_faulted_aem);
	
	timer_init(
		object_name					:= CONCAT(prc_path, 'connection_time_out_tmr'),
		process						:= prc,
		CONVERSION_this				:= connection_time_out_tmr);
		
	phase_init(
        object_name 				:= CONCAT(prc_path, '_cam_change_check_ph'),
        phase 						:= 0,	//Set at runtime!
        delay 						:= 0,
        max_compensation 			:= 0,
        generator 					:= csp_transfer_accumulator_virtualMaster.phgen,
        process 					:= prc,
        CONVERSION_this 			:= cam_change_check_ph);
		
	motorization_conditioner_init(
		object_name					:=	CONCAT(prc_path, 'connection_done_motcond'),
		velocity_limit				:=	0.0,
		velocity_limit_active		:=	FALSE,
		idle_handshake_active		:=	FALSE,
		execute_handshake_active	:=	TRUE,
		hold_handshake_active		:=	FALSE,
		suspend_handshake_active	:=	FALSE,
		complete_handshake_active	:=	FALSE,
		abort_handshake_active		:=	FALSE,
		stop_handshake_active		:=	FALSE,
		origin						:=	MOTORIZATION_CONDITIONER_ORIGIN_INTERNAL,
		manager						:=	csp_main_motorization_manager.motm,
		process						:=	prc,
		CONVERSION_this				:=	connection_done_motcond);
	
		
END_IF

IF objects_running()
THEN
	process_cycle(prc);
	
	axis_cycle(axis);
	
	phase_cycle(cam_change_check_ph);
	
	motorization_conditioner_cycle(connection_done_motcond);
	
END_IF
END_ACTION

ACTION _read_process_image:
;
END_ACTION

ACTION _read_var_input:
;
END_ACTION

ACTION _set_runtime_properties:
axis_actual_position := axis_get_actual_modulo_position(axis);
enable_delay(IN:=axis_is_ready_to_enable(axis) , PT:=T#2S , Q=> servo_on_condition , ET=> );
(* Cam management *)
IF 	connection_done
THEN
	active_cam := axis.engaged_cam.cam_id;
END_IF
END_ACTION

ACTION _write_output:
;
END_ACTION

ACTION connection:
connection_conditions :=	
	axis_is_ok(FALSE, axis)
	AND
	servo_on_condition
	AND
	NOT process_message_is_on(connection_faulted_aem)
	AND
	phase_done;

(* connection_done reset *)
IF	connection_done
	AND	
	NOT connection_conditions
	AND
	NOT csp.o_machine_is_running
THEN
	connection_done := FALSE;
END_IF

(* Exit conditions *)
IF	NOT connection_conditions
THEN	
	connection_status_next := CSP_TRANSFER_ACCUMULATOR_STATUS_CONNECTION_ERROR;
	connection_status := connection_status_next;	
END_IF

(*************** MACHINE STATUS ***************)
CASE connection_status OF

	CSP_TRANSFER_ACCUMULATOR_STATUS_CONNECTION_START:	(* Start connection *)
	
		IF	motorization_manager_is_starting(csp_main_motorization_manager.motm) //TODOPZ: da decidere a che livello usare le variabili di i e o: wn_feeding.i_motorization_is_starting?					
		THEN
			connection_running := TRUE;
			connection_status_next := CSP_TRANSFER_ACCUMULATOR_STATUS_CONNECTION_ENGAGE;
		END_IF
		
		
	CSP_TRANSFER_ACCUMULATOR_STATUS_CONNECTION_ENGAGE:	
	
		master_offset := axis_get_actual_modulo_position(csp_transfer_accumulator_virtualMaster.axis);			

		axis_engage_cam(
			cam_id							:=	active_cam,	
			master_engage_mode				:=	AXIS_CAM_ENGAGE_RELATIVE,
			slave_engage_mode				:=	AXIS_CAM_ENGAGE_RELATIVE,
			activation_mode					:=	AXIS_CAM_ACTIVATION_IMMEDIATELY,
			activation_position				:=	0.0,
			master_scaling_mode				:=	AXIS_CAM_SCALING_MODE_USER_DEFINED,
			slave_scaling_mode				:=	AXIS_CAM_SCALING_MODE_AUTOOFFSET,
			master_offset					:=	0, 
			slave_offset					:=	0.0,
			master_scaling					:=	master_scaling,
			slave_scaling					:=	slave_scaling,
			interpolation_type				:=	AXIS_CAM_INTERPOLATION_SPLINE,	 
			master							:=	csp_transfer_accumulator_virtualMaster.axis,
			CONVERSION_this					:=	axis);
		
		connection_status_next:= CSP_TRANSFER_ACCUMULATOR_STATUS_CONNECTION_ENGAGED;
	
		
	CSP_TRANSFER_ACCUMULATOR_STATUS_CONNECTION_ENGAGED:
	
		IF active_cam = 0
		THEN
			active_cam := next_cam;
		END_IF	
	
		IF 	axis_is_cam_engaged(axis) 
		THEN				
			IF	active_cam <> next_cam
			THEN							
				connection_status_next := CSP_TRANSFER_ACCUMULATOR_STATUS_CONNECTION_CHANGE_CAM;
			ELSE
				connection_status_next:= CSP_TRANSFER_ACCUMULATOR_STATUS_CONNECTION_DONE;
			END_IF
		END_IF
		
		
	CSP_TRANSFER_ACCUMULATOR_STATUS_CONNECTION_CHECK_CHANGE_CAM:	
		
		(* CARTONS AT BACKSTOP - NO NEED TO INDEX *)
	 	IF run
		THEN		
			CASE active_cam OF
			
				DWELL_CAM: 
					next_cam := TRANSFER_ACCUMULATOR_BELT_RUN;	
					run := FALSE;
					
				TRANSFER_ACCUMULATOR_BELT_RUN:
					run := FALSE;
					
			END_CASE			
		END_IF
	
		IF 	dwell
		THEN	
			
			CASE active_cam OF
				
				DWELL_CAM: 
					dwell := FALSE;				
					
				TRANSFER_ACCUMULATOR_BELT_RUN:
					next_cam := DWELL_CAM;
					dwell := FALSE;			
			END_CASE				
		END_IF		
		
		IF active_cam = TRANSFER_ACCUMULATOR_BELT_RUN
		THEN 
			next_cam := DWELL_CAM;
		END_IF		
		
		IF	active_cam <> next_cam
		THEN
			connection_status_next := CSP_TRANSFER_ACCUMULATOR_STATUS_CONNECTION_CHANGE_CAM;
		END_IF
		
		IF	NOT connection_motorization_moving
		THEN
			connection_status_next := CSP_TRANSFER_ACCUMULATOR_STATUS_CONNECTION_DONE;
		END_IF
	
		
	CSP_TRANSFER_ACCUMULATOR_STATUS_CONNECTION_CHANGE_CAM:	
	
		IF next_cam = TRANSFER_ACCUMULATOR_BELT_RUN
		THEN
			activation_mode := AXIS_CAM_ACTIVATION_IMMEDIATELY;
		ELSE
			activation_mode := AXIS_CAM_ACTIVATION_NEXT_CYCLE;
		END_IF
	
		axis_engage_cam(
				cam_id							:=	next_cam,	
				master_engage_mode				:=	AXIS_CAM_ENGAGE_RELATIVE,
				slave_engage_mode				:=	AXIS_CAM_ENGAGE_RELATIVE,
				activation_mode					:=	activation_mode,
				activation_position				:=	0,
				master_scaling_mode				:=	AXIS_CAM_SCALING_MODE_USER_DEFINED,
				slave_scaling_mode				:=	AXIS_CAM_SCALING_MODE_AUTOOFFSET,
				master_offset					:=	0, 
				slave_offset					:=	0.0,
				master_scaling					:=	master_scaling,
				slave_scaling					:=	slave_scaling,
				interpolation_type				:=	AXIS_CAM_INTERPOLATION_SPLINE,	 
				master							:=	csp_transfer_accumulator_virtualMaster.axis,
				CONVERSION_this					:=	axis);		
			
		IF	motorization_manager_is_starting(csp_main_motorization_manager.motm)
		THEN
			connection_status_next := CSP_TRANSFER_ACCUMULATOR_STATUS_CONNECTION_DONE;
		ELSE
			connection_status_next := CSP_TRANSFER_ACCUMULATOR_STATUS_CONNECTION_WAIT_NEW_CAM;
		END_IF
	
		
	CSP_TRANSFER_ACCUMULATOR_STATUS_CONNECTION_WAIT_NEW_CAM:
	
		IF	active_cam = next_cam
		THEN
			connection_status_next := CSP_TRANSFER_ACCUMULATOR_STATUS_CONNECTION_CHECK_CHANGE_CAM;
		END_IF
		
		IF	NOT connection_motorization_moving
		THEN
			connection_status_next := CSP_TRANSFER_ACCUMULATOR_STATUS_CONNECTION_DONE;
		END_IF
		
		
	CSP_TRANSFER_ACCUMULATOR_STATUS_CONNECTION_DONE:	(* Connection done *)	
	
		connection_running := FALSE;
		connection_done := TRUE;
		
		IF	motorization_manager_is_starting(csp_main_motorization_manager.motm)
		THEN
			motorization_conditioner_start_done(connection_done_motcond);
		END_IF
		connection_status_next := CSP_TRANSFER_ACCUMULATOR_STATUS_CONNECTION_CHECK_CHANGE_CAM;
	
		
	CSP_TRANSFER_ACCUMULATOR_STATUS_CONNECTION_ERROR:	(* Connection error *)	
	
		IF 	connection_running
			OR NOT axis_is_ok(FALSE, axis)
		THEN
			axis_disable(axis);	
			connection_error := TRUE;						
		END_IF
		connection_running	:= FALSE;
		connection_done 	:= FALSE;	
		
		IF	connection_conditions
		THEN		
			connection_status_next := CSP_TRANSFER_ACCUMULATOR_STATUS_CONNECTION_START;
		END_IF		
END_CASE

IF 	NOT debug_state_machine
	OR
	debug_connection_machine_one_step	
THEN
	connection_status := connection_status_next;
	debug_connection_machine_one_step := FALSE;
END_IF

connection_motorization_moving	:= 
	motorization_manager_is_starting(csp_main_motorization_manager.motm)
	OR
	motorization_manager_is_execute(csp_main_motorization_manager.motm)
	OR
	motorization_manager_is_stopping(csp_main_motorization_manager.motm)
	OR
	motorization_manager_is_suspended(csp_main_motorization_manager.motm)
	OR
	motorization_manager_is_suspending(csp_main_motorization_manager.motm)
	OR
	motorization_manager_is_unsuspending(csp_main_motorization_manager.motm)
	OR 
	motorization_manager_is_holding(csp_main_motorization_manager.motm)
	OR
	motorization_manager_is_held(csp_main_motorization_manager.motm)
	OR
	motorization_manager_is_unholding(csp_main_motorization_manager.motm);
	
(* Connection timeout *)
IF	(connection_running
	AND NOT debug_state_machine)	
	OR connection_error
THEN
	IF	timer_is_expired(connection_time_out_tmr)
	THEN
		process_message_set(1, connection_status, 0, connection_faulted_aem);
	END_IF
ELSE
	timer_restart(10000, connection_time_out_tmr);
END_IF
END_ACTION

ACTION phase:
phase_conditions :=
	axis_is_ok(FALSE, axis)
	AND
	process_is_ready(prc)
	AND
	process_subtree_is_ready(prc)
	AND
	servo_on_condition
	AND				
	NOT csp_transfer_main_brand.cam_data_changed
	AND
	NOT jog_manager_is_jog_axis_active(SMTR41323_TRANSFER_ACCUMULATOR_BELT, csp_main_jogManager.jog_manager_real)
	AND
	NOT disable_req;		
	
(* phase_done reset *)
IF	phase_done
	AND
	NOT phase_conditions
	AND 
	NOT csp.o_machine_is_running
THEN
	axis_disable(axis);
	
	phase_done:= FALSE;
END_IF

(* Exit condition *)
IF NOT phase_conditions
THEN
	phase_status_next := CSP_TRANSFER_ACCUMULATOR_BELT_STATUS_PHASE_ERROR;
	phase_status := phase_status_next;	
END_IF

(*************** MACHINE STATUS ***************)
CASE phase_status OF

	CSP_TRANSFER_ACCUMULATOR_BELT_STATUS_PHASE_START:	(* Start phasing *)
	
		IF	motorization_manager_is_starting(csp_main_motorization_manager.motm) 					
			AND axis_is_cam_engaged(csp_transfer_accumulator_virtualMaster.axis) (* Verifies the master is engaged before calculating position *)
		THEN
			phase_running := TRUE;
			phase_master_is_engaged := axis_is_cam_engaged(csp_transfer_accumulator_virtualMaster.axis);
			phase_status_next := CSP_TRANSFER_ACCUMULATOR_BELT_STATUS_PHASE_DISABLE;
		END_IF
						
	CSP_TRANSFER_ACCUMULATOR_BELT_STATUS_PHASE_DISABLE:
	
		axis_disable(axis);		
		
		IF 	axis_is_disabled(axis)
		THEN
			phase_status_next := CSP_TRANSFER_ACCUMULATOR_BELT_STATUS_PHASE_ENABLE;
		END_IF
		
		
	CSP_TRANSFER_ACCUMULATOR_BELT_STATUS_PHASE_ENABLE:
	
		axis_enable(axis);
		
		IF 	axis_is_enabled(axis)
		THEN
			phase_status_next := CSP_TRANSFER_ACCUMULATOR_BELT_STATUS_PHASE_ENABLED;
		END_IF
		
		
	CSP_TRANSFER_ACCUMULATOR_BELT_STATUS_PHASE_ENABLED:
	
		IF 	axis_is_standstill(axis) 
		THEN
			IF	phase_master_is_engaged
			THEN
				phase_status_next := CSP_TRANSFER_ACCUMULATOR_BELT_STATUS_PHASE_DONE;
			ELSE
				phase_status_next := CSP_TRANSFER_ACCUMULATOR_BELT_STATUS_PHASE_REDEFINE;
			END_IF					
		END_IF
		
		
	CSP_TRANSFER_ACCUMULATOR_BELT_STATUS_PHASE_REDEFINE:
	
		IF	axis_is_cam_engaged(csp_transfer_accumulator_virtualMaster.axis)
		THEN
			IF	axis_redefine_position(
					position			:= 0.0,
					mode				:= AXIS_REDEFINE_POSITION_MODE_ABSOLUTE,
					CONVERSION_this		:= axis)
			THEN
				phase_status_next := CSP_TRANSFER_ACCUMULATOR_BELT_STATUS_PHASE_REDEFINED;
			ELSE
				phase_status_next := CSP_TRANSFER_ACCUMULATOR_BELT_STATUS_PHASE_ERROR;
			END_IF
		END_IF
		
		
	CSP_TRANSFER_ACCUMULATOR_BELT_STATUS_PHASE_REDEFINED:
	
		IF 	axis_is_position_redefined(axis)
		THEN
			phase_status_next := CSP_TRANSFER_ACCUMULATOR_BELT_STATUS_PHASE_DONE;
		END_IF
		
		
	CSP_TRANSFER_ACCUMULATOR_BELT_STATUS_PHASE_DONE:	(* Phase done *)	
		
		phase_running := FALSE;
		phase_done := TRUE;				
	
		
	CSP_TRANSFER_ACCUMULATOR_BELT_STATUS_PHASE_ERROR:	(* Phase error *)
	
		IF	phase_running
		THEN
			phase_error := TRUE;
			axis_disable(axis);									
		END_IF
		phase_running := FALSE;
		
		IF	phase_conditions 	
		THEN
			phase_status_next := CSP_TRANSFER_ACCUMULATOR_BELT_STATUS_PHASE_START;
		END_IF
		
END_CASE

IF 	NOT debug_state_machine
	OR
	debug_phase_machine_one_step	
THEN
	phase_status := phase_status_next;
	debug_phase_machine_one_step := FALSE;
END_IF

(* Phasing timeout *)
IF	(phase_running
	AND NOT debug_state_machine)	
	OR phase_error
THEN
	IF	timer_is_expired(phase_time_out_tmr)
	THEN
		process_message_set(1, phase_status, 0, phase_faulted_aem);
	END_IF
ELSE
	timer_restart(10000, phase_time_out_tmr);
END_IF
END_ACTION

END_PROGRAM

// ---- Application/CSP/Transfer/Accumulator/csp_transfer_accumulator.TcPOU
(*********************************** G.D S.p.A. - Technical Department ***********************************
============= PROGRAM INFO ============
FOLDER:             TBD
MACHINES INVOLVED:  TBD 

============= DESCRIPTION =============
csp machine declaration

============= REVISIONS ===============
Date		Version	 	Author      	Description             
----------	-------		------------  	--------------------------------------------
2019/04/05 	0000.00	 	M.Grasso		Creation of the PRG

**********************************************************************************************************)
(*$R process_ref := prc; $*)
PROGRAM csp_transfer_accumulator
VAR
	
	prc:											process;
	prc_path:										STRING;
	
	index_request:									BOOL; (* Upstacker will set this to high when it picks up the cartons and begins route to fingers *)
	
	manual_index_belts:								BOOL;
	index_belts:									BOOL; 
	
	lift_not_cammed_dchk:							digital_check;
	lift_not_cammed_boolean:						boolean;
	
	upstacker_virtual_phgen:						phase_generator;
	upstacker_virtual_phwin:						phase_window; (* Used for the upstacker clear of cartons *)
	upstacker_cleared_cartons_low_limit:			LREAL := 20; (*$P $*)
	upstacker_cleared_cartons_high_limit:			LREAL := 30; (*$P $*)
	upstacker_clear:								BOOL;
	
END_VAR

_read_var_input();

_object_manager();

IF NOT objects_running()
THEN
	RETURN;	
END_IF

_read_process_image();

_mode_manager();

_set_runtime_properties();

(********************************* BODY *********************************)

(************************************************************************)

_handle_messages();

_write_output();

ACTION _handle_messages:
;
END_ACTION

ACTION _handle_process_test:
;
END_ACTION

ACTION _mode_manager:
IF process_mode_req_is_pending(prc)
THEN
    process_apply_mode_req_first_step(prc);
    CASE process_get_mode(prc) OF
        MODE_TO_ABSENT:
			;
        MODE_TO_INACTIVE:
			;
        MODE_TO_TEST:
			;
        MODE_TO_OPERATIONAL:
			;
    END_CASE
    process_apply_mode_req_second_step(prc);
END_IF
END_ACTION

ACTION _object_manager:
IF objects_initialization()
THEN
	sub_process_init(
		object_name					:= 'csp_transfer_accumulator.prc', 
		process						:= csp_transfer.prc, 
		CONVERSION_this				:= prc);
		
	prc_path 						:= process_get_path(prc);
	
	
	boolean_init(
		object_name:= CONCAT(prc_path, '_lift_not_cammed_boolean'), 
		process:= prc, 
		CONVERSION_this:= lift_not_cammed_boolean);
		
	digital_check_and_message_init(
		object_name:= CONCAT(prc_path, '_lift_not_cammed_dchk'), 
		alarm_if_input_off:= FALSE, 
		alarm_delay:= 2000, 
		enabled_at_powerup:= TRUE, 
		individual_reset:= FALSE, 
		machine_reaction:= MACHINE_REACTION_NORMAL_STOP, 
		typology:= MESSAGE_TYPOLOGY_ABNORMAL, 
		process:= prc, 
		CONVERSION_this:= lift_not_cammed_dchk);
		
	digital_check_add_boolean(
		boolean:= lift_not_cammed_boolean, 
		CONVERSION_this:= lift_not_cammed_dchk);
		
		
	(* PHASE GENERATORS *)
	phase_generator_init(
		object_name:= CONCAT(prc_path, '_upstacker_virtual_generator'), 
		modulo:= 360, 
		resolution:= PHASE_GENERATOR_RESOLUTION_UNIT, 
		axis:= csp_transfer_upstacker_virtualMaster.axis, 
		process:= prc, 
		CONVERSION_this:= upstacker_virtual_phgen);
		
	(* PHASE WINDOWS *)
	phase_window_init(
		object_name:= CONCAT(prc_path, '_upstacker_virtual_window'), 
		begin_phase:= upstacker_cleared_cartons_low_limit, 
		end_phase:= upstacker_cleared_cartons_high_limit, 
		begin_delay:= 0, 
		end_delay:= 0, 
		begin_max_compensation:= 0, 
		end_max_compensation:= 0, 
		generator:= upstacker_virtual_phgen, 
		process:= prc, 
		CONVERSION_this:= upstacker_virtual_phwin);		
	
END_IF

IF objects_running()
THEN
	process_cycle(prc);
	digital_check_cycle(lift_not_cammed_dchk);
	phase_generator_cycle(upstacker_virtual_phgen);	
	phase_window_cycle(upstacker_virtual_phwin);
	
END_IF
END_ACTION

ACTION _read_process_image:
;
END_ACTION

ACTION _read_var_input:
;
END_ACTION

ACTION _set_runtime_properties:
;
END_ACTION

ACTION _write_output:
;
END_ACTION

END_PROGRAM

// ---- Application/CSP/Transfer/csp_transfer.TcPOU
(*********************************** G.D S.p.A. - Technical Department ***********************************
============= PROGRAM INFO ============
FOLDER:             TBD
MACHINES INVOLVED:  TBD 

============= DESCRIPTION =============
csp machine declaration

============= REVISIONS ===============
Date		Version	 	Author      	Description             
----------	-------		------------  	--------------------------------------------
2019/04/05 	0000.00	 	M.Grasso		Creation of the PRG

**********************************************************************************************************)
(*$R process_ref := prc; $*)
PROGRAM csp_transfer
VAR
	
	prc:											process;
	prc_path:										STRING;
	
	disable_req:									BOOL;
	virtual_disable_req:							BOOL;
	
	disable_all_axes:								BOOL := FALSE; (*$P $*)
	manual_disable_all_axes:						BOOL := FALSE;
	
	transfer_cammed_motcond:						motorization_conditioner;
	
	PhaseOff_MainMoto_Transfer_VM: 					LREAL;
	PhaseOff_TransferVM_Crosspush_VM: 				LREAL;
	PhaseOff_TransferVM_Accumulator_VM: 			LREAL;
	Gear_TransferVM_AcculatorVM: 					LREAL;
	PhaseOff_AccumulatorVM_Upstacker_VM: 			LREAL;
END_VAR

_read_var_input();

_object_manager();

IF NOT objects_running()
THEN
	RETURN;	
END_IF

_read_process_image();

_mode_manager();

_set_runtime_properties();

(********************************* BODY *********************************)

(* MACHINE COMMANDS *)
IF csp_transfer_main_services_pushbuttons.reset_command
THEN
	machine_reset(csp.mch);
END_IF

IF csp_transfer_main_services_pushbuttons.start_command
THEN
	machine_start(csp.mch);
END_IF


(* Main disable request for real axes *)
disable_req := 	NOT machine_is_running(csp.mch)
				//OR
				//csp.i_reset_button
				//)
				//AND
				//process_is_ready(prc)
				AND machine_is_stop_emergency_active(csp.mch)
				AND csp_main_motorization_virtualManager.axis.actual_velocity = 0;

				
				
(* Verifies tranfer virtual is cam engaged and allows motorization to start *)
IF axis_is_cam_engaged(csp_transfer_virtualMaster.axis)
THEN
	motorization_conditioner_start_done(transfer_cammed_motcond);
ELSE
	motorization_conditioner_stop_done(transfer_cammed_motcond);
END_IF


IF csp_main_motorization.abort_axes
THEN
	disable_all_axes := TRUE;
END_IF


(* DISABLE VIRTUAL AXES *)
IF disable_all_axes
	OR manual_disable_all_axes
	OR
	(	
		( (* TRANSFER VIRTUAL MASTER CONNECTION DONE + PHASE DONE BUT DISABLED *)
			csp_transfer_virtualMaster.phase_done
			AND
			csp_transfer_virtualMaster.connection_done
			AND
			axis_is_disabled(csp_transfer_virtualMaster.axis)
		)
		OR
		( (* ACCUMULATOR VIRTUAL MASTER CONNECTION DONE + PHASE DONE BUT DISABLED *)
			csp_transfer_accumulator_virtualMaster.phase_done
			AND
			csp_transfer_accumulator_virtualMaster.connection_done
			AND
			axis_is_disabled(csp_transfer_accumulator_virtualMaster.axis)
		)
		OR
		( (* UPSTACKER VIRTUAL MASTER CONNECTION DONE + PHASE DONE BUT DISABLED *)
			csp_transfer_upstacker_virtualMaster.phase_done
			AND
			csp_transfer_upstacker_virtualMaster.connection_done
			AND
			axis_is_disabled(csp_transfer_upstacker_virtualMaster.axis)
		)
		OR
		( (* CROSSPUSHER VIRTUAL MASTER CONNECTION DONE + PHASE DONE BUT DISABLED *)
			csp_transfer_crosspusher_virtualMaster.phase_done
			AND
			csp_transfer_crosspusher_virtualMaster.connection_done
			AND
			axis_is_disabled(csp_transfer_crosspusher_virtualMaster.axis)
		)
	)
THEN
	disable_all_axes := FALSE;
	manual_disable_all_axes := FALSE;
	virtual_disable_req := TRUE;
ELSE
	virtual_disable_req := FALSE;
END_IF
		

(************************************************************************)

_handle_messages();

_write_output();

ACTION _handle_messages:
;
END_ACTION

ACTION _handle_process_test:
;
END_ACTION

ACTION _mode_manager:
IF process_mode_req_is_pending(prc)
THEN
    process_apply_mode_req_first_step(prc);
    CASE process_get_mode(prc) OF
        MODE_TO_ABSENT:
			;
        MODE_TO_INACTIVE:
			;
        MODE_TO_TEST:
			;
        MODE_TO_OPERATIONAL:
			;
    END_CASE
    process_apply_mode_req_second_step(prc);
END_IF
END_ACTION

ACTION _object_manager:
IF objects_initialization()
THEN
	process_init(
		object_name					:= 'csp_transfer.prc', 
		machine						:= csp.mch, 
		CONVERSION_this				:= prc);
		
	prc_path 						:= process_get_path(prc);
	
	
	motorization_conditioner_init(
		object_name								:=	CONCAT(prc_path, '_transfer_cammed_motcond'),
		velocity_limit							:=	100.0,
		velocity_limit_active					:=	FALSE,
		idle_handshake_active					:=	FALSE,
		execute_handshake_active				:=	FALSE,
		hold_handshake_active					:=	FALSE,
		suspend_handshake_active				:=	FALSE,
		complete_handshake_active				:=	FALSE,
		abort_handshake_active					:=	FALSE,
		stop_handshake_active					:=	FALSE,
		origin									:=	MOTORIZATION_CONDITIONER_ORIGIN_INTERNAL,
		manager									:=	csp_main_motorization_manager.motm,
		process									:=	prc,
		CONVERSION_this							:=	transfer_cammed_motcond);
	
END_IF

IF objects_running()
THEN
	process_cycle(prc);
	
	motorization_conditioner_cycle(transfer_cammed_motcond);
	
END_IF
END_ACTION

ACTION _read_process_image:
;
END_ACTION

ACTION _read_var_input:
;
END_ACTION

ACTION _set_runtime_properties:
;
END_ACTION

ACTION _write_output:
;
END_ACTION

END_PROGRAM

// ---- Application/CSP/Transfer/Virtual Master/csp_transfer_virtualMaster.TcPOU
(*********************************** G.D S.p.A. - Technical Department ***********************************
============= PROGRAM INFO ============
FOLDER:             TBD
MACHINES INVOLVED:  TBD 

============= DESCRIPTION =============
csp machine declaration

============= REVISIONS ===============
Date		Version	 	Author      	Description             
----------	-------		------------  	--------------------------------------------
2019/04/05 	0000.00	 	M.Grasso		Creation of the PRG

**********************************************************************************************************)
(*$R process_ref := prc; $*)
PROGRAM csp_transfer_virtualMaster
VAR
	
	prc:											process;
	prc_path:										STRING;
	
	fsm_enable_condition:							BOOL := FALSE;
	fsm_next_status:								csp_transfer_status_enum;
	fsm_status:										csp_transfer_status_enum;
	
	axis: 											axis;
	phgen:											phase_generator;
	tranfer_vm_phgen:								phase_generator;
	
	phase_position_deg:								LREAL := 0;
	phase_velocity_degps:							LREAL := 100.0;
	
	home_position_master_offset_deg:				LREAL := 0.0;
	axis_calculate_cam_slave_master_position_deg:	LREAL := 0.0;
	axis_calculated_cam_slave_position_deg:			LREAL := 0.0;	
	slave_position_has_been_calculated:				BOOL  := FALSE;
	
	phase_enable:									BOOL := TRUE;
	slave_position_request:							BOOL := TRUE;
	engage_enable:									BOOL := TRUE;
	
	cam_id:											DINT  := FORWARD_CAM;
	slave_scaling:									LREAL := 1.0 (*360.0*);
	master_scaling:									LREAL := 1.0 (*360.0*);
	master_cam:										LREAL := 30;
	
	master_offset_phase:							LREAL;
	
	transfer_running:								BOOL := TRUE;
	dwell:											BOOL;
	run:											BOOL;
	
	dwell_test:										BOOL;
	run_test:										BOOL;
	
	active_cam:										DINT := FORWARD_CAM;
	next_cam:										DINT := FORWARD_CAM;
	
	connection_status: 								csp_transfer_connection_status_enum;
	connection_status_next: 						csp_transfer_connection_status_enum;
	connection_done: 								BOOL;
	connection_running: 							BOOL;
	connection_error:								BOOL;
	connection_time_out_tmr:						timer;
	connection_faulted_aem:	 						message;
	connection_conditions:							BOOL;
	connection_done_motcond:						motorization_conditioner;
	connection_motorization_moving:					BOOL;
	
	next_activation_position:						LREAL;	
	activation_position:							LREAL := 0.0;
	
	
	phase_status: 									csp_transfer_phase_status_enum;
	phase_status_next: 								csp_transfer_phase_status_enum;
	phase_done: 									BOOL;
	phase_running: 									BOOL;
	phase_error:									BOOL;
	phase_time_out_tmr:								timer;
	phase_faulted_aem:	 							message;
	phase_conditions:								BOOL;
	phase_slave_position:							LREAL;
	
	section_0_180:									BOOL;	
	section_180_360:								BOOL;
	section_0_120:									BOOL;
	section_120_240:								BOOL;
	section_240_360:								BOOL;
	
	cam_change_check_ph:							phase;
	
	section_0_180_phwin:							phase_window;
	section_180_360_phwin:							phase_window;
	section_0_120_phwin:							phase_window;
	section_120_240_phwin:							phase_window;
	section_240_360_phwin:							phase_window;
	
	disable_req:									BOOL;
	debug_state_machine:							BOOL := FALSE;
	debug_phase_machine_one_step:					BOOL := FALSE;
	debug_connection_machine_one_step:				BOOL := FALSE;
	debug_immediate_stop_aem:						message;
	debug_immediate_stop:							BOOL;
	
	position_difference:							LREAL;
	position_difference_tolerance:					LREAL := 3;
	axis_off_from_offset_boolean:					boolean;
	axis_off_from_offset_aem:						message;
	
	Upstacker_Rephase_Clear_Product: 				message;
	Upstacker_Rephase_Verified: 					BOOL;
END_VAR

VAR CONSTANT
	
	MOTOR_MAX_VELOCITY_DEGPS:						LREAL := 9600;
	MOTOR_MAX_ACCELERATION_DEGPS2:					LREAL := 48000;
	MOTOR_MAX_DECELERATION_DEGPS2:					LREAL := 48000;
	MOTOR_MAX_JERK_DEGPS3:							LREAL := 1000000; 
	MOTOR_MAX_FOLLOWING_ERROR_DEG:					LREAL := 2;
	
	CAM_CHANGE_CHECK_DEG:							LREAL := 350;

END_VAR

_read_var_input();

_object_manager();

IF NOT objects_running()
THEN
	RETURN;	
END_IF

_read_process_image();

_mode_manager();

CASE process_get_mode(prc) OF
	MODE_ABSENT,
	MODE_INACTIVE:
		RETURN;
	MODE_TEST:
		_handle_process_test();
END_CASE

(********************************* BODY *********************************)
phase_set_data(
	phase				:= CAM_CHANGE_CHECK_DEG,
	delay				:= 0,			
	max_compensation	:= 0,			
	CONVERSION_this		:= cam_change_check_ph);
	
	
(* USES MASTER OFFSET OF LOADER PUSHER SINCE IT MUST SYNC WITH IT AT ALL TIMES TO LOAD *)
home_position_master_offset_deg := csp_case_loader_virtualMaster.home_position_master_offset_deg;
	
	
IF phase_edge(cam_change_check_ph)
THEN
	IF run_test 
	OR 
	(
		NOT csp_transfer_crosspusher.reject_dwell_transfer
		OR NOT csp_transfer_upstacker_sensors.dwell_transfer_empty
		OR 
		(
			csp_transfer_crosspusher.reject_done
			AND
			csp_case_loader_virtualMaster.loader_finishing_after_reject
			AND														 
			axis_is_cam_engaged(csp_transfer_crosspusher_horizontal.axis)
			AND
			axis_is_cam_engaged(csp_transfer_crosspusher_vertical.axis)
			AND
			axis_is_cam_engaged(csp_transfer_crosspusher_follower.axis)
		)
	)
	THEN
		dwell := FALSE;
		run := TRUE;
	ELSE
		dwell := TRUE;
		run := FALSE;
	END_IF
END_IF


(* Connection Done *)
IF connection_done
THEN 
	motorization_conditioner_start_done(connection_done_motcond);
END_IF


(* RESETS AXES IF PHASE DONE AND CONNECTION DONE AND DISABLED *)
IF 	phase_done
	AND connection_done
	AND axis_is_disabled(axis)
THEN
	phase_done := FALSE;
	connection_done := FALSE;
END_IF


jog_manager_set_all_slave_axis_engaged(
	index					:= JOG_LIST_TRANSFER_VIRTUAL, 
	all_slave_axis_engaged	:= 	axis_is_cam_engaged(csp_transfer_accumulator_virtualMaster.axis)
							 	AND
							 	axis_is_cam_engaged(csp_transfer_crosspusher_virtualMaster.axis),
	CONVERSION_this			:= csp_main_jogManager.jog_manager_virtual);


(* DISABLES VIRTUAL IS ANY OF THE SLAVES FAULT *)
IF 	NOT axis_is_disabled(axis)
	AND NOT axis_is_ok(FALSE, csp_transfer_crosspusher_virtualMaster.axis)
	AND NOT axis_is_ok(FALSE, csp_transfer_accumulator_virtualMaster.axis)
THEN
	axis_disable(axis);
END_IF


(* DOESN'T ALLOW FOR CAM TO EVER BE 0 *)
IF 	active_cam = 0
THEN 
	active_cam := DWELL_CAM;
END_IF


(* CLEARS PHASE AND CONNECTION ERRORS ON STOP *)
IF 	machine_is_stopped(csp.mch)
	OR machine_is_stop_emergency_active(csp.mch)
THEN
	phase_error := FALSE;
	connection_error := FALSE;	
END_IF


(* CHECKS THAT THE TRANSFER IS NOT OFF FROM ITS POSITION *)
position_difference := LMOD(360, ABS(axis.actual_position - csp_main_motorization_virtualManager.axis.actual_position) - home_position_master_offset_deg);

IF 	active_cam = FORWARD_CAM
	AND position_difference > position_difference_tolerance
	AND csp_transfer_virtualMaster.phase_done
	AND machine_is_running(csp.mch)
THEN
	;
ELSE
	;
END_IF


(* SETS ALL PHASE WINDOWS FOR SECTIONS BASED ON COUNT *)
section_0_180 := phase_window_position_is_in_window(axis.actual_position, section_0_180_phwin);
section_180_360 := phase_window_position_is_in_window(axis.actual_position, section_180_360_phwin);
section_0_120 := phase_window_position_is_in_window(axis.actual_position, section_0_120_phwin);
section_120_240 := phase_window_position_is_in_window(axis.actual_position, section_120_240_phwin);
section_240_360 := phase_window_position_is_in_window(axis.actual_position, section_240_360_phwin);


(* PHASE DATA FOR 0 TO 180 *)
phase_window_set_phases_data(
	begin_phase					:= 0,
	end_phase					:= 180,
	begin_delay					:= 0,
	end_delay					:= 0,
	begin_max_compensation		:= 0,
	end_max_compensation		:= 0,
	CONVERSION_this				:= section_0_180_phwin);
	
(* PHASE DATA FOR 180 TO 359.999 *)
phase_window_set_phases_data(
	begin_phase					:= 180,
	end_phase					:= 359.999,
	begin_delay					:= 0,
	end_delay					:= 0,
	begin_max_compensation		:= 0,
	end_max_compensation		:= 0,
	CONVERSION_this				:= section_180_360_phwin);
	
(* PHASE DATA FOR 0 TO 120 *)
phase_window_set_phases_data(
	begin_phase					:= 0,
	end_phase					:= 120,
	begin_delay					:= 0,
	end_delay					:= 0,
	begin_max_compensation		:= 0,
	end_max_compensation		:= 0,
	CONVERSION_this				:= section_0_120_phwin);
	
(* PHASE DATA FOR 120 TO 240 *)
phase_window_set_phases_data(
	begin_phase					:= 120,
	end_phase					:= 240,
	begin_delay					:= 0,
	end_delay					:= 0,
	begin_max_compensation		:= 0,
	end_max_compensation		:= 0,
	CONVERSION_this				:= section_120_240_phwin);
	
(* PHASE DATA FOR 240 TO 359.999 *)
phase_window_set_phases_data(
	begin_phase					:= 240,
	end_phase					:= 359.999,
	begin_delay					:= 0,
	end_delay					:= 0,
	begin_max_compensation		:= 0,
	end_max_compensation		:= 0,
	CONVERSION_this				:= section_240_360_phwin);


phase();
connection();
_set_runtime_properties();
(************************************************************************)

_handle_messages();

_write_output();

ACTION _handle_messages:
IF process_message_is_on(Upstacker_Rephase_Clear_Product) 
	AND NOT csp_transfer_main_safety_guards.sis.is_safely_closed 
THEN
	Upstacker_Rephase_Verified := TRUE;
	process_message_reset(Upstacker_Rephase_Clear_Product);
END_IF
END_ACTION

ACTION _handle_process_test:
;
END_ACTION

ACTION _mode_manager:
IF process_mode_req_is_pending(prc)
THEN
    process_apply_mode_req_first_step(prc);
    CASE process_get_mode(prc) OF
        MODE_TO_ABSENT:
			;
        MODE_TO_INACTIVE:
			;
        MODE_TO_TEST:
			;
        MODE_TO_OPERATIONAL:
			;
    END_CASE
    process_apply_mode_req_second_step(prc);
END_IF
END_ACTION

ACTION _object_manager:
IF objects_initialization()
THEN
	sub_process_init(
		object_name					:= 'csp_transfer_virtualMaster.prc', 
		process						:= csp_transfer.prc, 
		CONVERSION_this				:= prc);
		
	prc_path 						:= process_get_path(prc);
	
	axis_init(
		object_name					:= CONCAT(prc_path, '_axis'), 
		axis_type					:= AXIS_TYPE_VIRTUAL, 
		encoder_scaling_factor		:= G_VIRTUAL_ENCODER_SCALING_FACTOR_DEGPINC,
		modulo						:= G_MODULO_360_DEG, 
		process						:= prc, 
		CONVERSION_this				:= axis);
	
	axis_set_max_dynamic(
		reference_velocity			:=	MOTOR_MAX_VELOCITY_DEGPS,
		velocity					:=	MOTOR_MAX_VELOCITY_DEGPS,
		acceleration				:=	MOTOR_MAX_ACCELERATION_DEGPS2,
		deceleration				:=	MOTOR_MAX_DECELERATION_DEGPS2,
		jerk						:=	MOTOR_MAX_JERK_DEGPS3,
		following_error				:=	MOTOR_MAX_FOLLOWING_ERROR_DEG,
		CONVERSION_this				:=	axis);
		
	phase_generator_init(
		object_name					:= CONCAT(prc_path, '_phgen'), 
		modulo						:= axis_get_modulo(axis), 
		resolution					:= PHASE_GENERATOR_RESOLUTION_UNIT, 
		axis						:= axis, 
		process						:= prc, 
		CONVERSION_this				:= phgen);
		
		
	phase_init(
        object_name 				:= CONCAT(prc_path, '_cam_change_check_ph'),
        phase 						:= 0,	//Set at runtime!
        delay 						:= 0,
        max_compensation 			:= 0,
        generator 					:= phgen,
        process 					:= prc,
        CONVERSION_this 			:= cam_change_check_ph);
		
	process_message_init(
		object_name					:=	CONCAT(prc_path, '_phase_faulted_aem'), 
		behaviour					:=	MESSAGE_BEHAVIOUR_EVENT,
		reset_timeout				:=	0,
		disableable					:=	TRUE,
		individual_reset			:=	FALSE,
		machine_reaction			:=	MACHINE_REACTION_NORMAL_STOP,
		typology					:=	MESSAGE_TYPOLOGY_ABNORMAL,
		process						:=	prc,
		CONVERSION_this				:=	phase_faulted_aem);
	
	timer_init(
		object_name					:= CONCAT(prc_path, 'phase_time_out_tmr'),
		process						:= prc,
		CONVERSION_this				:= phase_time_out_tmr);
		
	process_message_init(
		object_name					:=	CONCAT(prc_path, 'debug_immediate_stop_aem'), 
		behaviour					:=	MESSAGE_BEHAVIOUR_STATE,
		reset_timeout				:=	0,
		disableable					:=	TRUE,
		individual_reset			:=	FALSE,
		machine_reaction			:=	MACHINE_REACTION_NORMAL_STOP,
		typology					:=	MESSAGE_TYPOLOGY_ABNORMAL,
		process						:=	prc,
		CONVERSION_this				:=	debug_immediate_stop_aem);
		
	timer_init(
		object_name					:= CONCAT(prc_path, 'connection_time_out_tmr'),
		process						:= prc,
		CONVERSION_this				:= connection_time_out_tmr);
		
		
	process_message_init(
		object_name					:=	CONCAT(prc_path, '_connection_faulted_aem'), 
		behaviour					:=	MESSAGE_BEHAVIOUR_EVENT,
		reset_timeout				:=	0,
		disableable					:=	TRUE,
		individual_reset			:=	FALSE,
		machine_reaction			:=	MACHINE_REACTION_NORMAL_STOP,
		typology					:=	MESSAGE_TYPOLOGY_ABNORMAL,
		process						:=	prc,
		CONVERSION_this				:=	connection_faulted_aem);
		
	motorization_conditioner_init(
		object_name					:=	CONCAT(prc_path, 'connection_done_motcond'),
		velocity_limit				:=	0.0,
		velocity_limit_active		:=	FALSE,
		idle_handshake_active		:=	FALSE,
		execute_handshake_active	:=	TRUE,
		hold_handshake_active		:=	FALSE,
		suspend_handshake_active	:=	FALSE,
		complete_handshake_active	:=	FALSE,
		abort_handshake_active		:=	FALSE,
		stop_handshake_active		:=	FALSE,
		origin						:=	MOTORIZATION_CONDITIONER_ORIGIN_INTERNAL,
		manager						:=	csp_main_motorization_manager.motm,
		process						:=	prc,
		CONVERSION_this				:=	connection_done_motcond);
		
	phase_window_init(
		object_name					:= CONCAT(prc_path, '_section_0_180_phwin'), 
		begin_phase					:= 0, 
		end_phase					:= 180, 
		begin_delay					:= 0, 
		end_delay					:= 0, 
		begin_max_compensation		:= 0, 
		end_max_compensation		:= 0, 
		generator					:= phgen, 
		process						:= prc, 
		CONVERSION_this				:= section_0_180_phwin);
	
	phase_window_init(
		object_name					:= CONCAT(prc_path, '_section_180_360_phwin'), 
		begin_phase					:= 180, 
		end_phase					:= 359.999, 
		begin_delay					:= 0, 
		end_delay					:= 0, 
		begin_max_compensation		:= 0, 
		end_max_compensation		:= 0, 
		generator					:= phgen, 
		process						:= prc, 
		CONVERSION_this				:= section_180_360_phwin);
		
	phase_window_init(
		object_name					:= CONCAT(prc_path, '_section_0_120_phwin'), 
		begin_phase					:= 0, 
		end_phase					:= 120, 
		begin_delay					:= 0, 
		end_delay					:= 0, 
		begin_max_compensation		:= 0, 
		end_max_compensation		:= 0, 
		generator					:= phgen, 
		process						:= prc, 
		CONVERSION_this				:= section_0_120_phwin);
		
	phase_window_init(
		object_name					:= CONCAT(prc_path, '_section_120_240_phwin'), 
		begin_phase					:= 120, 
		end_phase					:= 240, 
		begin_delay					:= 0, 
		end_delay					:= 0, 
		begin_max_compensation		:= 0, 
		end_max_compensation		:= 0, 
		generator					:= phgen, 
		process						:= prc, 
		CONVERSION_this				:= section_120_240_phwin);
		
	phase_window_init(
		object_name					:= CONCAT(prc_path, '_section_240_360_phwin'), 
		begin_phase					:= 240, 
		end_phase					:= 359.999, 
		begin_delay					:= 0, 
		end_delay					:= 0, 
		begin_max_compensation		:= 0, 
		end_max_compensation		:= 0, 
		generator					:= phgen, 
		process						:= prc, 
		CONVERSION_this				:= section_240_360_phwin);
		
		
	jog_manager_add_axis(
		list_index					:= JOG_LIST_TRANSFER_VIRTUAL,
		axis						:= axis,
		master_axis					:= TRUE,
		jog_type					:= JOG_TYPE_ROTATIVE,
		sw_limit_positive			:= 0,
		sw_limit_negative			:= 0,
		CONVERSION_this				:= csp_main_jogManager.jog_manager_virtual);
		
		
		
	process_message_init(
		object_name					:=	CONCAT(prc_path, '_axis_off_from_offset_aem'), 
		behaviour					:=	MESSAGE_BEHAVIOUR_EVENT,
		reset_timeout				:=	0,
		disableable					:=	FALSE,
		individual_reset			:=	FALSE,
		machine_reaction			:=	MACHINE_REACTION_STOP_IN_PHASE_ONE,
		typology					:=	MESSAGE_TYPOLOGY_ABNORMAL,
		process						:=	prc,
		CONVERSION_this				:=	axis_off_from_offset_aem);
	
	process_message_init(
		object_name					:=	CONCAT(prc_path, '_Upstacker_Rephase_Clear_Product'), 
		behaviour					:=	MESSAGE_BEHAVIOUR_EVENT,
		reset_timeout				:=	0,
		disableable					:=	TRUE,
		individual_reset			:=	TRUE,
		machine_reaction			:=	MACHINE_REACTION_NORMAL_STOP,
		typology					:=	MESSAGE_TYPOLOGY_ABNORMAL,
		process						:=	prc,
		CONVERSION_this				:=	Upstacker_Rephase_Clear_Product);

END_IF

IF objects_running()
THEN
	process_cycle(prc);
	motorization_conditioner_cycle(connection_done_motcond);
	
	axis_cycle(axis);
	phase_generator_cycle(phgen);
	phase_cycle(cam_change_check_ph);
	
	phase_window_cycle(section_0_180_phwin);
	phase_window_cycle(section_180_360_phwin);
	phase_window_cycle(section_0_120_phwin);
	phase_window_cycle(section_120_240_phwin);
	phase_window_cycle(section_240_360_phwin);
END_IF
END_ACTION

ACTION _read_process_image:
;
END_ACTION

ACTION _read_var_input:
disable_req := csp_transfer.virtual_disable_req;
END_ACTION

ACTION _set_runtime_properties:
(* Cam management *)
IF 	connection_done
THEN
	active_cam := axis.engaged_cam.cam_id;
END_IF
END_ACTION

ACTION _write_output:
;
END_ACTION

ACTION connection:
connection_conditions :=	
	NOT process_message_is_on(connection_faulted_aem)
	//AND
	//NOT jog_manager_is_jog_axis_active(JOG_LIST_TRANSFER_VIRTUAL, csp_main_jogManager.jog_manager_virtual)
	AND
	phase_done;

(* connection_done reset *)
IF	connection_done
	AND	
	NOT connection_conditions
	AND
	NOT csp.o_machine_is_running
THEN
	connection_done := FALSE;
END_IF

(* Exit conditions *)
IF	NOT connection_conditions 
	AND
	NOT motorization_manager_is_stopping(csp_main_motorization_manager.motm)	
THEN	
	connection_status_next := CSP_TRANSFER_STATUS_CONNECTION_ERROR;
	connection_status := connection_status_next;	
END_IF

(*************** MACHINE STATUS ***************)
CASE connection_status OF

	CSP_TRANSFER_STATUS_CONNECTION_START:	(* Start connection *)
		IF	motorization_manager_is_starting(csp_main_motorization_manager.motm) //TODOPZ: da decidere a che livello usare le variabili di i e o: wn_feeding.i_motorization_is_starting?					
		THEN
			connection_running := TRUE;
			connection_status_next := CSP_TRANSFER_STATUS_CONNECTION_ENGAGE;
		END_IF
		
	CSP_TRANSFER_STATUS_CONNECTION_ENGAGE:		
	
		master_offset_phase := csp_main_motorization_virtualManager.axis.actual_modulo_position;	
			
		axis_engage_cam(
			cam_id							:=	active_cam,	
			master_engage_mode				:=	AXIS_CAM_ENGAGE_RELATIVE,
			slave_engage_mode				:=	AXIS_CAM_ENGAGE_RELATIVE,
			activation_mode					:=	AXIS_CAM_ACTIVATION_IMMEDIATELY,
			activation_position				:=	0.0,
			master_scaling_mode				:=	AXIS_CAM_SCALING_MODE_USER_DEFINED,
			slave_scaling_mode				:=	AXIS_CAM_SCALING_MODE_AUTOOFFSET,
			master_offset					:=	LMOD(home_position_master_offset_deg + master_offset_phase, axis_get_modulo(csp_main_motorization_virtualManager.axis)),
			slave_offset					:=	0.0,
			master_scaling					:=	master_scaling,
			slave_scaling					:=	slave_scaling,
			interpolation_type				:=	AXIS_CAM_INTERPOLATION_SPLINE,	 
			master							:=	csp_main_motorization_virtualManager.axis,
			CONVERSION_this					:=	axis);
		
		connection_status_next:= CSP_TRANSFER_STATUS_CONNECTION_ENGAGED;
	
	CSP_TRANSFER_STATUS_CONNECTION_ENGAGED:
	
		IF active_cam = 0
		THEN
			active_cam := next_cam;
		END_IF
	
		IF 	axis_is_cam_engaged(axis) 
		THEN				
			IF	active_cam <> next_cam
			THEN							
				connection_status_next := CSP_TRANSFER_STATUS_CONNECTION_CHANGE_CAM;
			ELSE
				connection_status_next:= CSP_TRANSFER_STATUS_CONNECTION_DONE;
			END_IF
		END_IF
		
	CSP_TRANSFER_STATUS_CONNECTION_CHECK_CHANGE_CAM:						
		IF dwell
		THEN
			next_cam := DWELL_CAM;
			dwell:= FALSE;
		END_IF
				
		IF run
		THEN
			next_cam := FORWARD_CAM;
			run := FALSE;
		END_IF	
		
		IF	(active_cam <> next_cam)
			AND 
			connection_conditions
		THEN							
			connection_status_next := CSP_TRANSFER_STATUS_CONNECTION_CHANGE_CAM;
		END_IF
			
		IF	NOT connection_motorization_moving
		THEN
			connection_status_next := CSP_TRANSFER_STATUS_CONNECTION_DONE;
		END_IF
	
	CSP_TRANSFER_STATUS_CONNECTION_CHANGE_CAM:	
		
		axis_engage_cam(
				cam_id							:=	next_cam,	
				master_engage_mode				:=	AXIS_CAM_ENGAGE_ABSOLUTE,
				slave_engage_mode				:=	AXIS_CAM_ENGAGE_RELATIVE,
				activation_mode					:=	AXIS_CAM_ACTIVATION_NEXT_CYCLE,
				activation_position				:=	0,
				master_scaling_mode				:=	AXIS_CAM_SCALING_MODE_USER_DEFINED,
				slave_scaling_mode				:=	AXIS_CAM_SCALING_MODE_USER_DEFINED,
				master_offset					:=	home_position_master_offset_deg, 
				slave_offset					:=	0.0,
				master_scaling					:=	master_scaling,
				slave_scaling					:=	slave_scaling,
				interpolation_type				:=	AXIS_CAM_INTERPOLATION_SPLINE,	 
				master							:=	csp_main_motorization_virtualManager.axis,
				CONVERSION_this					:=	axis);	
	
		IF	motorization_manager_is_starting(csp_main_motorization_manager.motm)
		THEN
			connection_status_next := CSP_TRANSFER_STATUS_CONNECTION_DONE;
		ELSE
			IF axis_is_cam_engaged(axis)
			THEN
				connection_status_next := CSP_TRANSFER_STATUS_CONNECTION_WAIT_NEW_CAM;
			END_IF
		END_IF
	
	CSP_TRANSFER_STATUS_CONNECTION_WAIT_NEW_CAM:
		IF	active_cam = next_cam
		THEN
			CASE next_cam OF
				DWELL_CAM:
					activation_position := next_activation_position;
				
				FORWARD_CAM:
					activation_position := 0;
					
			END_CASE
			connection_status_next := CSP_TRANSFER_STATUS_CONNECTION_CHECK_CHANGE_CAM;
		END_IF
		
		IF	NOT connection_motorization_moving
		THEN
			connection_status_next := CSP_TRANSFER_STATUS_CONNECTION_DONE;
		END_IF
		
	CSP_TRANSFER_STATUS_CONNECTION_DONE:	(* Connection done *)		
		connection_running := FALSE;
		connection_done := TRUE;
		
		IF	motorization_manager_is_starting(csp_main_motorization_manager.motm)
		THEN
			motorization_conditioner_start_done(connection_done_motcond);							
			IF	active_cam <> next_cam
			THEN
				connection_status_next := CSP_TRANSFER_STATUS_CONNECTION_WAIT_NEW_CAM;
			ELSE
				connection_status_next := CSP_TRANSFER_STATUS_CONNECTION_CHECK_CHANGE_CAM;
			END_IF
		END_IF
	
	CSP_TRANSFER_STATUS_CONNECTION_ERROR:	(* Connection error *)	
		IF 	connection_running
		THEN
			axis_disable(axis);
			connection_error := TRUE;						
		END_IF
		connection_running	:= FALSE;
		connection_done 	:= FALSE;	
		
		IF	connection_conditions
		THEN		
			connection_status_next := CSP_TRANSFER_STATUS_CONNECTION_START;
		END_IF
		
END_CASE

IF 	NOT debug_state_machine
	OR
	debug_connection_machine_one_step	
THEN
	connection_status := connection_status_next;
	debug_connection_machine_one_step := FALSE;
END_IF

connection_motorization_moving	:= 
	motorization_manager_is_starting(csp_main_motorization_manager.motm)
	OR
	motorization_manager_is_execute(csp_main_motorization_manager.motm)
	OR
	motorization_manager_is_stopping(csp_main_motorization_manager.motm)	
	//OR
	//csp_main_motorization_manager.motm.actual_velocity > 0 
	OR
	motorization_manager_is_suspended(csp_main_motorization_manager.motm)
	OR
	motorization_manager_is_suspending(csp_main_motorization_manager.motm)
	OR
	motorization_manager_is_unsuspending(csp_main_motorization_manager.motm)
	OR
	motorization_manager_is_holding(csp_main_motorization_manager.motm)
	OR
	motorization_manager_is_held(csp_main_motorization_manager.motm)
	OR
	motorization_manager_is_unholding(csp_main_motorization_manager.motm);
	
(* Connection timeout *)
IF	(connection_running
	AND NOT debug_state_machine)	
	OR connection_error
THEN
	IF	timer_is_expired(connection_time_out_tmr)
	THEN
		process_message_set(1, connection_status, 0, connection_faulted_aem);
	END_IF
ELSE
	timer_restart(10000, connection_time_out_tmr);
END_IF
END_ACTION

ACTION phase:
phase_conditions :=
	axis_is_ok(FALSE, axis)
	AND
	process_is_ready(prc)
	AND
	process_subtree_is_ready(prc)
	AND				
	NOT csp_transfer_main_brand.cam_data_changed
	AND
	NOT jog_manager_is_jog_axis_active(JOG_LIST_TRANSFER_VIRTUAL, csp_main_jogManager.jog_manager_virtual)
	AND
	NOT disable_req;		
	
(* phase_done reset *)
IF	phase_done
	AND
	NOT phase_conditions
THEN
	phase_done:= FALSE;
END_IF

(* Exit condition *)
IF 	NOT phase_conditions
THEN
	phase_status_next := CSP_TRANSFER_PHASE_STATUS_ERROR;
	phase_status := phase_status_next;	
END_IF

(*************** MACHINE STATUS ***************)
CASE phase_status OF

	CSP_TRANSFER_PHASE_STATUS_START:	(* Start phasing *)
		IF	motorization_manager_is_starting(csp_main_motorization_manager.motm) //TODOPZ: da decidere a che livello usare le variabili di i e o: wn_feeding.i_motorization_is_starting?					
		THEN
			phase_running := TRUE;			
			phase_status_next := CSP_TRANSFER_PHASE_STATUS_DISABLE;
		END_IF
						
	CSP_TRANSFER_PHASE_STATUS_DISABLE:
		axis_disable(axis);		
		
		IF 	axis_is_disabled(axis)
		THEN
			phase_status_next := CSP_TRANSFER_PHASE_STATUS_ENABLE;
		END_IF
		
	CSP_TRANSFER_PHASE_STATUS_ENABLE:
		axis_enable(axis);
		
		IF 	axis_is_enabled(axis)
		THEN
			phase_status_next := CSP_TRANSFER_PHASE_STATUS_ENABLED;
		END_IF
		
	CSP_TRANSFER_PHASE_STATUS_ENABLED:
		IF 	axis_is_standstill(axis) 
		THEN
			phase_status_next := CSP_TRANSFER_PHASE_STATUS_CALCULATE_SLAVE_POSITION_REQUEST;								
		END_IF
		
	CSP_TRANSFER_PHASE_STATUS_CALCULATE_SLAVE_POSITION_REQUEST:
		slave_position_has_been_calculated := FALSE;
	
		(* Gets the position of the master axis *)
		axis_calculate_cam_slave_master_position_deg := 
			LMOD(axis_get_actual_modulo_position(csp_main_motorization_virtualManager.axis)
			+ home_position_master_offset_deg, G_MODULO_360_DEG);
			
		(* Gets cam data for slave axis to master *)
		IF axis_calculate_cam_slave_dynamics_data(
			cam_id := active_cam,
			master_scaling := master_scaling,
			master_position := axis_calculate_cam_slave_master_position_deg,
			slave_scaling := slave_scaling,
			CONVERSION_this := csp_transfer_virtualMaster.axis)
		THEN
			phase_status_next := CSP_TRANSFER_PHASE_STATUS_CALCULATING_SLAVE_POSITION;
		END_IF
	
	CSP_TRANSFER_PHASE_STATUS_CALCULATING_SLAVE_POSITION:
		IF axis_cam_slave_dynamics_data_calculated(csp_transfer_virtualMaster.axis)
		THEN
			axis_calculated_cam_slave_position_deg := axis_get_cam_slave_dynamics_position(csp_transfer_virtualMaster.axis);
			slave_position_has_been_calculated := TRUE;
			phase_status_next := CSP_TRANSFER_PHASE_STATUS_REQUEST;
				
		END_IF
		
	CSP_TRANSFER_PHASE_STATUS_REQUEST:
		IF	axis_is_standstill(axis)
		(* RMH - MAYBE have to wait for slave axes to cam *)
		
		THEN
		 axis_move_absolute(
			position 		:= axis_calculated_cam_slave_position_deg,
			velocity 		:= phase_velocity_degps,
			direction		:= AXIS_SHORTEST_WAY,
			acceleration 	:= MOTOR_MAX_ACCELERATION_DEGPS2,
			deceleration 	:= MOTOR_MAX_DECELERATION_DEGPS2, 
			jerk 			:= MOTOR_MAX_JERK_DEGPS3, 
			buffer_mode 	:= AXIS_BUFFER_MODE_BUFFERED,
			CONVERSION_this := axis
			); 
		END_IF

		IF axis_is_absolute_moving(axis)
		THEN
			phase_status_next	:=	CSP_TRANSFER_PHASE_STATUS_PHASING;
		END_IF

	CSP_TRANSFER_PHASE_STATUS_PHASING:
		IF axis_is_standstill(axis)
		THEN
			phase_status_next	:=	CSP_TRANSFER_STATUS_PHASED;
		END_IF

	CSP_TRANSFER_STATUS_PHASED:
		IF engage_enable
		THEN
			phase_status_next := CSP_TRANSFER_PHASE_STATUS_DONE;
		END_IF
		
		
	CSP_TRANSFER_PHASE_STATUS_DONE:	(* Phase done *)			
		phase_running := FALSE;
		phase_done := TRUE;				
	
	CSP_TRANSFER_PHASE_STATUS_ERROR:	(* Phase error *)
		IF	phase_running
		THEN
			phase_error := TRUE;
			axis_disable(axis);									
		END_IF
		phase_running := FALSE;
		
		IF	phase_conditions 	
		THEN
			phase_status_next := CSP_TRANSFER_PHASE_STATUS_START;
		END_IF
		
END_CASE

IF 	NOT debug_state_machine
	OR
	debug_phase_machine_one_step	
THEN
	phase_status := phase_status_next;
	debug_phase_machine_one_step := FALSE;
END_IF

(* Phasing timeout *)
IF (phase_running
	AND NOT debug_state_machine)
	OR phase_error
THEN
	IF	timer_is_expired(phase_time_out_tmr)
	THEN
		process_message_set(1, phase_status, 0, phase_faulted_aem);
	END_IF
ELSE
	timer_restart(10000, phase_time_out_tmr);
END_IF
END_ACTION

END_PROGRAM

// ---- Application/CSP/Case/Loader/Virtual Master/csp_case_loader_virtualMaster.TcPOU
(*********************************** G.D S.p.A. - Technical Department ***********************************
============= PROGRAM INFO ============
FOLDER:             TBD
MACHINES INVOLVED:  TBD 

============= DESCRIPTION =============
csp machine declaration

============= REVISIONS ===============
Date		Version	 	Author      	Description             
----------	-------		------------  	--------------------------------------------
2019/04/05 	0000.00	 	M.Grasso		Creation of the PRG

**********************************************************************************************************)
(*$R process_ref := prc; $*)
PROGRAM csp_case_loader_virtualMaster
VAR
	
	
	prc:												process;
	prc_path:											STRING;
	
	fsm_enable_condition:								BOOL := FALSE;
	fsm_next_status:									CSP_CASE_LOADER_STATUS_enum;
	fsm_status:											CSP_CASE_LOADER_STATUS_enum;
	phase_enable:										BOOL  := TRUE;
	axis: 												axis;
	
	phase_position_deg:									LREAL := 0;
	phase_velocity_degps:								LREAL := 20.0;
	axis_calculate_cam_slave_master_position_deg:		LREAL := 0.0;
	axis_calculated_cam_slave_position_deg:				LREAL := 0.0;
	slave_position_has_been_calculated:					BOOL  := FALSE;
	engage_enable:										BOOL:=TRUE;
	disable_req:										BOOL:=FALSE;
	debug_state_machine:								BOOL:=FALSE;
	debug_state_machine_one_step:						BOOL:=FALSE;
 
	master_offset_phase:								LREAL;
	
	
	cam_id:												DINT  := LINEAR_CAM;	
	slave_scaling_mm:									LREAL := 1; 
	master_scaling_deg:									LREAL := 1; 
	slave_scaling:										LREAL := 1; 
	master_scaling:										LREAL := 1; 
	home_position_master_offset_deg: 					LREAL := 240;
	loader_slaves_cammed:								BOOL  := FALSE;
	pusher_tolerance:									LREAL:= 5;
	
	target_position:									LREAL;
	
	product_loaded:										BOOL;
	product_pushing:									BOOL;
	case_loaded_chksect:								check_section;
	case_loaded_bool:									boolean;
	stop:												BOOL:= FALSE;
	master_offset: 										LREAL := 240;
	master_engage_mode:									axis_cam_engage_mode_enum;
	slave_offset: 										LREAL := 0;

	At_Reject_product_loaded: 							BOOL := FALSE;
	engage_after_estop: 								BOOL := FALSE;
	
	load_check_ph: 										phase;
	phgen:												phase_generator;
	load_check_deg: 									LREAL := 110;
	
	product_load_failed: 								BOOLean;
	product_load_failed_dchk: 							digital_check;
	phase_done: 										BOOL := FALSE;
	
	loader_run_check_ph:								phase;
	loader_run_check_deg:								LREAL; (* AUTO CALCULATED BASED ON LOADER PUSHER OFFSET *)
	loader_run_check_before_deg:						LREAL := 10;
	
	loader_finishing_after_reject:						BOOL;
	
	
	(* PHASE AND CONNECTION TEST *)
	connection_status: 									csp_case_connection_status_enum;
	connection_status_next: 							csp_case_connection_status_enum;
	connection_done: 									BOOL;
	connection_running: 								BOOL;
	connection_error:									BOOL;
	connection_time_out_tmr:							timer;
	connection_faulted_aem:	 							message;
	connection_conditions:								BOOL;
	connection_done_motcond:							motorization_conditioner;
	connection_motorization_moving:						BOOL;
	
	next_activation_position:							LREAL;	
	activation_position:								LREAL := 0.0;
	connection_status1: 								LREAL;
	connection_status_next1: 							LREAL;
	
	phase_status: 										csp_case_phase_status_enum;
	phase_status_next: 									csp_case_phase_status_enum;
	phase_running: 										BOOL;
	phase_error:										BOOL;
	phase_time_out_tmr:									timer;
	phase_faulted_aem:	 								message;
	phase_conditions:									BOOL;
	phase_slave_position:								LREAL;
	
	debug_phase_machine_one_step:						BOOL := FALSE;
	debug_connection_machine_one_step:					BOOL := FALSE;
	debug_immediate_stop_aem:							message;
	debug_immediate_stop:								BOOL;
	
	active_cam:											DINT := DWELL_CAM;
	next_cam:											DINT := DWELL_CAM;
	
	dwell:												BOOL;
	run:												BOOL;
	
	Engagement_Error_aem: 								message;
	engage_count: INT := 0;
END_VAR

VAR CONSTANT
	
	CONSTANTS:											csp_case_loader_constant_struct;

END_VAR

_read_var_input();

_object_manager();

IF NOT objects_running()
THEN
	RETURN;	
END_IF

_read_process_image();

_mode_manager();

CASE process_get_mode(prc) of
	MODE_ABSENT,
	MODE_INACTIVE:
		RETURN;
	MODE_TEST:
		_handle_process_test();
END_CASE


(********************************* BODY *********************************)
connection_status1 := connection_status;
connection_status_next1 := connection_status_next; 

(*FSM Control*)
(*disable_req := NOT machine_is_running(csp.mch)
                AND machine_is_stop_emergency_active(csp.mch)
                AND csp_main_motorization_virtualManager.axis.actual_velocity = 0;*)	//_read_var_input
				
IF 	axis_is_cam_engaged(csp_case_loader_guide_downstream.axis)
	//AND axis_is_cam_engaged(csp_case_loader_guide_length.axis)
	AND axis_is_cam_engaged(csp_case_loader_guide_upstream.axis)
	AND axis_is_cam_engaged(csp_case_loader_pusher.axis)
	//AND axis_is_cam_engaged(csp_case_fc_ls_lower_Trailingcloser.axis)
	//AND axis_is_cam_engaged(csp_case_fc_ls_upper_LeadingMinorCloser.axis)
THEN
	loader_slaves_cammed := TRUE;
ELSE
	loader_slaves_cammed := FALSE;	
END_IF

IF 	NOT csp_case_main_safety_emergency.sis.safely_closed_input.status 
	AND axis_is_cam_engaged(axis) 
THEN
	engage_after_estop := TRUE;
ELSIF csp_case_main_safety_emergency.sis.safely_closed_input.status 
	AND fsm_status = CSP_CASE_TRANSPORT_STATUS_CAM_ENGAGED 
THEN
		engage_after_estop := FALSE;
END_IF


(* PHASE USED TO CHECK AT 0 IF THE STACK WILL BE AT THE LOADER - NOT A DEFINITE STACK - GUESSING THAT IT MAKES IT THROUGH CROSSPUSH LIGHT CURTAIN *)
phase_set_data(
	phase				:= load_check_deg,
	delay				:= 0,			
	max_compensation	:= 0,			
	CONVERSION_this		:= load_check_ph);
	
	
(* PHASE TO CHECK RIGHT BEFORE LOADER PUSHER THAT THE STACK IS STILL AT LOADER BASED ON LIGHT CURTAIN *)
loader_run_check_deg := (360 - csp_case_loader_pusher.master_offset - loader_run_check_before_deg);

phase_set_data(
	phase				:= loader_run_check_deg,
	delay				:= 0,			
	max_compensation	:= 0,			
	CONVERSION_this		:= loader_run_check_ph);

	
(* SETS A BIT HIGH OF PRODUCT BEING PUSHED BY LOADER PUSHER *)
IF 	machine_is_running(csp.mch)
	AND csp_transfer_upstacker.stack_at_loader
	AND axis_is_moving(axis) //product was loaded if pos > 150 //dont check when not moving (startup)
THEN
	product_pushing := TRUE;
	At_Reject_product_loaded :=TRUE;
END_IF


(* IF PRODUCT IS BEING PUSHED BY LOADER PUSHER AND REACHES END OF STROKE - TURN PRODUCT LOADED TO HIGH AND NO LONGER BEING PUSHED *)
IF 	machine_is_running(csp.mch)
	AND product_pushing
	AND (ABS(csp_case_loader_pusher.axis.actual_position - csp_case_loader_pusher.slave_scaling) < pusher_tolerance) 
THEN
	product_loaded := TRUE;
	product_pushing := FALSE;
END_IF


(* IF THE PRODUCT IS STILL BEING PUSHED WHEN THE LOADER PUSHER RETURNS TO HOME POSITION THEN ERROR LOADING PRODUCT *)
IF 	machine_is_running(csp.mch)
	AND csp_case_virtualMaster.axis.actual_position < 5
THEN
	IF product_pushing
	THEN
		//boolean_set(product_load_failed);
	END_IF
		
	product_loaded := FALSE;
	product_pushing := FALSE;
END_IF

IF 	machine_is_stopped(csp.mch)
	OR machine_is_stop_emergency_active(csp.mch)
THEN
	boolean_reset(product_load_failed);
END_IF


IF	At_Reject_product_loaded 
	AND axis_is_moving(csp_case_transport_os_trailing.axis) 
THEN
	At_Reject_product_loaded := FALSE;
END_IF


IF 	csp_transfer_upstacker.stack_in_case_at_loader
	AND NOT csp_case_main_services.dry_cycle_mode
THEN
	boolean_set(case_loaded_bool);
ELSE
	boolean_reset(case_loaded_bool);
END_IF

(* NEW LOGIC TO CONTROL RUN - USING PHASE/CONNECTION *)
(* DECIDES WHETHER TO START OR STOP THE CASE VIRTUAL *)
IF 	phase_edge(load_check_ph)
THEN
		
	IF 
	( (* NORMAL OPERATION *)
		//csp_case_loader.cases_primed // CASE PRESENT AT STATION BEFORE LOAD
		csp_case_loader.case_at_loader // CASES PRESENT AT LOADER IN TRANSPORT
		AND csp_transfer_upstacker.stack_at_loader // STACK IS AT LOADER FROM CROSSPUSHER
		AND NOT csp_transfer_crosspusher_sensors.no_load_bool.status 
		AND NOT csp_transfer_upstacker.stack_in_case_at_loader // STACK IS NOT ALREADY IN THE CASE IN TRANSPORT
		AND NOT csp_case_transport_virtualMaster.stop_for_reject
		AND NOT csp_case_fc_ls_upper_leadingMinorCloser.at_upstream_pos
		AND NOT csp_transfer_crosspusher.reject_running // 6_30_2022
	)
	OR 
	( (* IN CASE JOGH IS ACTIVE TO RUN *)
		jog_manager_is_jog_axis_active(JOG_LIST_CSP_CASE_VIRTUAL, csp_main_jogManager.jog_manager_virtual)
	)
	THEN
		dwell := FALSE;
		run := TRUE;
	ELSE
		run := FALSE;
		dwell := TRUE;
	END_IF
		
END_IF


(* Connection Done *)
IF 	connection_done
THEN 
	motorization_conditioner_start_done(connection_done_motcond);
END_IF


(* RESETS AXES IF PHASE DONE AND CONNECTION DONE AND DISABLED *)
IF 	phase_done
	AND connection_done
	AND axis_is_disabled(axis)
THEN
	phase_done := FALSE;
	connection_done := FALSE;
END_IF


(* DISABLES VIRTUAL IS ANY OF THE SLAVES FAULT *)
IF 	NOT axis_is_disabled(axis)
	AND NOT axis_is_ok(FALSE, csp_case_loader_pusher.axis)
	AND NOT axis_is_ok(FALSE, csp_case_loader_guide_upstream.axis)
	AND NOT axis_is_ok(FALSE, csp_case_loader_guide_downstream.axis)
	AND NOT axis_is_ok(FALSE, csp_case_fc_ls_upper_leadingMinorCloser.axis)
	AND NOT axis_is_ok(FALSE, csp_case_fc_ls_lower_trailingCloser.axis)
THEN
	; //axis_disable(axis);
END_IF


(* CLEARS PHASE AND CONNECTION ERRORS ON STOP *)
IF 	machine_is_stopped(csp.mch)
	OR machine_is_stop_emergency_active(csp.mch)
THEN
	phase_error := FALSE;
	connection_error := FALSE;	
END_IF


phase();
connection();
_set_runtime_properties();

(*IF 	active_cam = 0
	OR 
	(
		(csp_transfer_crosspusher_sensors.reject_stack OR csp_transfer_crosspusher.reject_running)
		AND  active_cam <> DWELL_CAM
		AND csp_transfer_crosspusher.loader_clear
	)
THEN
		active_cam := DWELL_CAM;
END_IF
*)

IF 	csp_transfer_crosspusher_horizontal.axis.actual_position < -5
	AND axis_is_moving(axis)
	AND axis_is_cam_engaged(axis)
THEN
	process_message_set(1, 0, 0, Engagement_Error_aem);
ELSE
	process_message_reset(Engagement_Error_aem);
END_IF


(************************************************************************)

_handle_messages();

_write_output();

ACTION _handle_messages:
;
END_ACTION

ACTION _handle_process_test:
;
END_ACTION

ACTION _mode_manager:
IF process_mode_req_is_pending(prc)
THEN
    process_apply_mode_req_first_step(prc);
    CASE process_get_mode(prc) OF
        MODE_TO_ABSENT:
			;
        MODE_TO_INACTIVE:
			;
        MODE_TO_TEST:
			;
        MODE_TO_OPERATIONAL:
			;
    END_CASE
    process_apply_mode_req_second_step(prc);
END_IF
END_ACTION

ACTION _object_manager:
IF objects_initialization()
THEN
	sub_process_init(
		object_name					:= 'csp_case_loader_virtualMaster.prc', 
		process						:= csp_case_loader.prc, 
		CONVERSION_this				:= prc);
		
	prc_path 						:= process_get_path(prc);
	
